	CONST robtarget p717:=[[0.0000,-127.8373,13.7328],[0.0000,-0.0467,0.9989,0.0000],[-1,0,-1,0],[9E+09,0.0000,-489.6442,9E+09,9E+09,9E+09]];
	CONST robtarget p718:=[[0.0000,-127.6671,13.7523],[0.0000,-0.0390,0.9992,0.0000],[-1,0,-1,0],[9E+09,0.0000,-490.5328,9E+09,9E+09,9E+09]];
	CONST robtarget p719:=[[0.0000,-127.5276,13.7719],[0.0000,-0.0312,0.9995,0.0000],[-1,0,-1,0],[9E+09,0.0000,-491.4237,9E+09,9E+09,9E+09]];
	CONST robtarget p720:=[[0.0000,-127.4190,13.7914],[0.0000,-0.0234,0.9997,0.0000],[-1,0,-1,0],[9E+09,0.0000,-492.3162,9E+09,9E+09,9E+09]];
	CONST robtarget p721:=[[0.0000,-127.3414,13.8109],[0.0000,-0.0156,0.9999,0.0000],[-1,0,-1,0],[9E+09,0.0000,-493.2101,9E+09,9E+09,9E+09]];
	CONST robtarget p722:=[[0.0000,-127.2948,13.8305],[0.0000,-0.0078,1.0000,0.0000],[-1,0,-1,0],[9E+09,0.0000,-494.1048,9E+09,9E+09,9E+09]];
	CONST robtarget p723:=[[0.0000,-127.2792,13.8500],[0.0000,-0.0000,-1.0000,0.0000],[-1,0,-1,0],[9E+09,0.0000,-495.0000,9E+09,9E+09,9E+09]];
	CONST robtarget p724:=[[0.0000,-127.2948,13.8695],[0.0000,-0.0078,-1.0000,0.0000],[-1,0,-1,0],[9E+09,0.0000,-495.8952,9E+09,9E+09,9E+09]];
	CONST robtarget p725:=[[0.0000,-127.3414,13.8891],[0.0000,-0.0156,-0.9999,0.0000],[-1,0,-1,0],[9E+09,0.0000,-496.7899,9E+09,9E+09,9E+09]];
	CONST robtarget p726:=[[0.0000,-127.4190,13.9086],[0.0000,-0.0234,-0.9997,0.0000],[-1,0,-1,0],[9E+09,0.0000,-497.6838,9E+09,9E+09,9E+09]];
	CONST robtarget p727:=[[0.0000,-127.5276,13.9281],[0.0000,-0.0312,-0.9995,0.0000],[-1,0,-1,0],[9E+09,0.0000,-498.5763,9E+09,9E+09,9E+09]];
	CONST robtarget p728:=[[0.0000,-127.6671,13.9477],[0.0000,-0.0390,-0.9992,0.0000],[-1,0,-1,0],[9E+09,0.0000,-499.4672,9E+09,9E+09,9E+09]];
	CONST robtarget p729:=[[0.0000,-127.8373,13.9672],[0.0000,-0.0467,-0.9989,0.0000],[-1,0,-1,0],[9E+09,0.0000,-500.3558,9E+09,9E+09,9E+09]];
	CONST robtarget p730:=[[0.0000,-128.0383,13.9867],[0.0000,-0.0544,-0.9985,0.0000],[-1,0,-1,0],[9E+09,0.0000,-501.2419,9E+09,9E+09,9E+09]];
	CONST robtarget p731:=[[0.0000,-128.2697,14.0062],[0.0000,-0.0621,-0.9981,0.0000],[-1,0,-1,0],[9E+09,0.0000,-502.1250,9E+09,9E+09,9E+09]];
	CONST robtarget p732:=[[0.0000,-128.5316,14.0258],[0.0000,-0.0698,-0.9976,0.0000],[-1,0,-1,0],[9E+09,0.0000,-503.0047,9E+09,9E+09,9E+09]];
	CONST robtarget p733:=[[0.0000,-128.8236,14.0453],[0.0000,-0.0774,-0.9970,0.0000],[-1,0,-1,0],[9E+09,0.0000,-503.8807,9E+09,9E+09,9E+09]];
	CONST robtarget p734:=[[0.0000,-129.1455,14.0648],[0.0000,-0.0850,-0.9964,0.0000],[-1,0,-1,0],[9E+09,0.0000,-504.7524,9E+09,9E+09,9E+09]];
	CONST robtarget p735:=[[0.0000,-129.4972,14.0844],[0.0000,-0.0925,-0.9957,0.0000],[-1,0,-1,0],[9E+09,0.0000,-505.6197,9E+09,9E+09,9E+09]];
	CONST robtarget p736:=[[0.0000,-129.8784,14.1039],[0.0000,-0.1000,-0.9950,0.0000],[-1,0,-1,0],[9E+09,0.0000,-506.4820,9E+09,9E+09,9E+09]];
	CONST robtarget p737:=[[0.0000,-130.2889,14.1234],[0.0000,-0.1075,-0.9942,0.0000],[-1,0,-1,0],[9E+09,0.0000,-507.3391,9E+09,9E+09,9E+09]];
	CONST robtarget p738:=[[0.0000,-130.7283,14.1430],[0.0000,-0.1149,-0.9934,0.0000],[-1,0,-1,0],[9E+09,0.0000,-508.1906,9E+09,9E+09,9E+09]];
	CONST robtarget p739:=[[0.0000,-131.1964,14.1625],[0.0000,-0.1222,-0.9925,0.0000],[-1,0,-1,0],[9E+09,0.0000,-509.0362,9E+09,9E+09,9E+09]];
	CONST robtarget p740:=[[0.0000,-131.6929,14.1820],[0.0000,-0.1295,-0.9916,0.0000],[-1,0,-1,0],[9E+09,0.0000,-509.8757,9E+09,9E+09,9E+09]];
	CONST robtarget p741:=[[0.0000,-132.2174,14.2016],[0.0000,-0.1367,-0.9906,0.0000],[-1,0,-1,0],[9E+09,0.0000,-510.7086,9E+09,9E+09,9E+09]];
	CONST robtarget p742:=[[0.0000,-132.7697,14.2211],[0.0000,-0.1438,-0.9896,0.0000],[-1,0,-1,0],[9E+09,0.0000,-511.5348,9E+09,9E+09,9E+09]];
	CONST robtarget p743:=[[0.0000,-133.3493,14.2406],[0.0000,-0.1509,-0.9886,0.0000],[-1,0,-1,0],[9E+09,0.0000,-512.3540,9E+09,9E+09,9E+09]];
	CONST robtarget p744:=[[0.0000,-133.9559,14.2602],[0.0000,-0.1579,-0.9875,0.0000],[-1,0,-1,0],[9E+09,0.0000,-513.1660,9E+09,9E+09,9E+09]];
	CONST robtarget p745:=[[0.0000,-134.5892,14.2797],[0.0000,-0.1648,-0.9863,0.0000],[-1,0,-1,0],[9E+09,0.0000,-513.9704,9E+09,9E+09,9E+09]];
	CONST robtarget p746:=[[0.0000,-135.2488,14.2992],[0.0000,-0.1716,-0.9852,0.0000],[-1,0,-1,0],[9E+09,0.0000,-514.7672,9E+09,9E+09,9E+09]];
	CONST robtarget p747:=[[0.0000,-135.9343,14.3187],[0.0000,-0.1784,-0.9840,0.0000],[-1,0,-1,0],[9E+09,0.0000,-515.5560,9E+09,9E+09,9E+09]];
	CONST robtarget p748:=[[0.0000,-136.6452,14.3383],[0.0000,-0.1851,-0.9827,0.0000],[-1,0,-1,0],[9E+09,0.0000,-516.3369,9E+09,9E+09,9E+09]];
	CONST robtarget p749:=[[0.0000,-137.3813,14.3578],[0.0000,-0.1917,-0.9814,0.0000],[-1,0,-1,0],[9E+09,0.0000,-517.1094,9E+09,9E+09,9E+09]];
	CONST robtarget p750:=[[0.0000,-138.1421,14.3773],[0.0000,-0.1983,-0.9801,0.0000],[-1,0,-1,0],[9E+09,0.0000,-517.8737,9E+09,9E+09,9E+09]];
	CONST robtarget p751:=[[0.0000,-138.9273,14.3969],[0.0000,-0.2047,-0.9788,0.0000],[-1,0,-1,0],[9E+09,0.0000,-518.6294,9E+09,9E+09,9E+09]];
	CONST robtarget p752:=[[0.0000,-139.7363,14.4164],[0.0000,-0.2111,-0.9775,0.0000],[-1,0,-1,0],[9E+09,0.0000,-519.3765,9E+09,9E+09,9E+09]];
	CONST robtarget p753:=[[0.0000,-140.5687,14.4359],[0.0000,-0.2174,-0.9761,0.0000],[-1,0,-1,0],[9E+09,0.0000,-520.1148,9E+09,9E+09,9E+09]];
	CONST robtarget p754:=[[0.0000,-141.4243,14.4555],[0.0000,-0.2236,-0.9747,0.0000],[-1,0,-1,0],[9E+09,0.0000,-520.8444,9E+09,9E+09,9E+09]];
	CONST robtarget p755:=[[0.0000,-142.3025,14.4750],[0.0000,-0.2298,-0.9732,0.0000],[-1,0,-1,0],[9E+09,0.0000,-521.5651,9E+09,9E+09,9E+09]];
	CONST robtarget p756:=[[0.0000,-143.2029,14.4945],[0.0000,-0.2358,-0.9718,0.0000],[-1,0,-1,0],[9E+09,0.0000,-522.2768,9E+09,9E+09,9E+09]];
	CONST robtarget p757:=[[0.0000,-144.1252,14.5141],[0.0000,-0.2417,-0.9703,0.0000],[-1,0,-1,0],[9E+09,0.0000,-522.9795,9E+09,9E+09,9E+09]];
	CONST robtarget p758:=[[0.0000,-145.0688,14.5336],[0.0000,-0.2476,-0.9689,0.0000],[-1,0,-1,0],[9E+09,0.0000,-523.6731,9E+09,9E+09,9E+09]];
	CONST robtarget p759:=[[0.0000,-146.0335,14.5531],[0.0000,-0.2534,-0.9674,0.0000],[-1,0,-1,0],[9E+09,0.0000,-524.3578,9E+09,9E+09,9E+09]];
	CONST robtarget p760:=[[0.0000,-147.0187,14.5727],[0.0000,-0.2591,-0.9659,0.0000],[-1,0,-1,0],[9E+09,0.0000,-525.0333,9E+09,9E+09,9E+09]];
	CONST robtarget p761:=[[0.0000,-148.0241,14.5922],[0.0000,-0.2647,-0.9643,0.0000],[-1,0,-1,0],[9E+09,0.0000,-525.6997,9E+09,9E+09,9E+09]];
	CONST robtarget p762:=[[0.0000,-149.0492,14.6117],[0.0000,-0.2702,-0.9628,0.0000],[-1,0,-1,0],[9E+09,0.0000,-526.3571,9E+09,9E+09,9E+09]];
	CONST robtarget p763:=[[0.0000,-150.0937,14.6312],[0.0000,-0.2757,-0.9612,0.0000],[-1,0,-1,0],[9E+09,0.0000,-527.0054,9E+09,9E+09,9E+09]];
	CONST robtarget p764:=[[0.0000,-151.1572,14.6508],[0.0000,-0.2810,-0.9597,0.0000],[-1,0,-1,0],[9E+09,0.0000,-527.6446,9E+09,9E+09,9E+09]];
	CONST robtarget p765:=[[0.0000,-152.2391,14.6703],[0.0000,-0.2863,-0.9581,0.0000],[-1,0,-1,0],[9E+09,0.0000,-528.2749,9E+09,9E+09,9E+09]];
	CONST robtarget p766:=[[0.0000,-153.3393,14.6898],[0.0000,-0.2915,-0.9566,0.0000],[-1,0,-1,0],[9E+09,0.0000,-528.8962,9E+09,9E+09,9E+09]];
	CONST robtarget p767:=[[0.0000,-154.4572,14.7094],[0.0000,-0.2966,-0.9550,0.0000],[-1,0,-1,0],[9E+09,0.0000,-529.5085,9E+09,9E+09,9E+09]];
	CONST robtarget p768:=[[0.0000,-155.5925,14.7289],[0.0000,-0.3016,-0.9534,0.0000],[-1,0,-1,0],[9E+09,0.0000,-530.1120,9E+09,9E+09,9E+09]];
	CONST robtarget p769:=[[0.0000,-156.7448,14.7484],[0.0000,-0.3066,-0.9518,0.0000],[-1,0,-1,0],[9E+09,0.0000,-530.7067,9E+09,9E+09,9E+09]];
	CONST robtarget p770:=[[0.0000,-157.9138,14.7680],[0.0000,-0.3114,-0.9503,0.0000],[-1,0,-1,0],[9E+09,0.0000,-531.2926,9E+09,9E+09,9E+09]];
	CONST robtarget p771:=[[0.0000,-159.0990,14.7875],[0.0000,-0.3162,-0.9487,0.0000],[-1,0,-1,0],[9E+09,0.0000,-531.8699,9E+09,9E+09,9E+09]];
	CONST robtarget p772:=[[0.0000,-160.3002,14.8070],[0.0000,-0.3209,-0.9471,0.0000],[-1,0,-1,0],[9E+09,0.0000,-532.4386,9E+09,9E+09,9E+09]];
	CONST robtarget p773:=[[0.0000,-161.5169,14.8266],[0.0000,-0.3256,-0.9455,0.0000],[-1,0,-1,0],[9E+09,0.0000,-532.9987,9E+09,9E+09,9E+09]];
	CONST robtarget p774:=[[0.0000,-162.7488,14.8461],[0.0000,-0.3301,-0.9439,0.0000],[-1,0,-1,0],[9E+09,0.0000,-533.5505,9E+09,9E+09,9E+09]];
	CONST robtarget p775:=[[0.0000,-163.9955,14.8656],[0.0000,-0.3346,-0.9424,0.0000],[-1,0,-1,0],[9E+09,0.0000,-534.0939,9E+09,9E+09,9E+09]];
	CONST robtarget p776:=[[0.0000,-165.2568,14.8852],[0.0000,-0.3390,-0.9408,0.0000],[-1,0,-1,0],[9E+09,0.0000,-534.6290,9E+09,9E+09,9E+09]];
	CONST robtarget p777:=[[0.0000,-166.5323,14.9047],[0.0000,-0.3433,-0.9392,0.0000],[-1,0,-1,0],[9E+09,0.0000,-535.1560,9E+09,9E+09,9E+09]];
	CONST robtarget p778:=[[0.0000,-167.8217,14.9242],[0.0000,-0.3475,-0.9377,0.0000],[-1,0,-1,0],[9E+09,0.0000,-535.6749,9E+09,9E+09,9E+09]];
	CONST robtarget p779:=[[0.0000,-169.1246,14.9437],[0.0000,-0.3517,-0.9361,0.0000],[-1,0,-1,0],[9E+09,0.0000,-536.1859,9E+09,9E+09,9E+09]];
	CONST robtarget p780:=[[0.0000,-170.4407,14.9633],[0.0000,-0.3558,-0.9345,0.0000],[-1,0,-1,0],[9E+09,0.0000,-536.6891,9E+09,9E+09,9E+09]];
	CONST robtarget p781:=[[0.0000,-171.7699,14.9828],[0.0000,-0.3599,-0.9330,0.0000],[-1,0,-1,0],[9E+09,0.0000,-537.1844,9E+09,9E+09,9E+09]];
	CONST robtarget p782:=[[0.0000,-173.1116,15.0023],[0.0000,-0.3638,-0.9315,0.0000],[-1,0,-1,0],[9E+09,0.0000,-537.6722,9E+09,9E+09,9E+09]];
	CONST robtarget p783:=[[0.0000,-174.4657,15.0219],[0.0000,-0.3677,-0.9299,0.0000],[-1,0,-1,0],[9E+09,0.0000,-538.1524,9E+09,9E+09,9E+09]];
	CONST robtarget p784:=[[0.0000,-175.8319,15.0414],[0.0000,-0.3716,-0.9284,0.0000],[-1,0,-1,0],[9E+09,0.0000,-538.6252,9E+09,9E+09,9E+09]];
	CONST robtarget p785:=[[0.0000,-177.2098,15.0609],[0.0000,-0.3753,-0.9269,0.0000],[-1,0,-1,0],[9E+09,0.0000,-539.0906,9E+09,9E+09,9E+09]];
	CONST robtarget p786:=[[0.0000,-178.5993,15.0805],[0.0000,-0.3790,-0.9254,0.0000],[-1,0,-1,0],[9E+09,0.0000,-539.5489,9E+09,9E+09,9E+09]];
	CONST robtarget p787:=[[0.0000,-180.0000,15.1000],[0.0000,-0.3827,0.9239,0.0000],[-1,0,-1,0],[9E+09,0.0000,-540.0000,9E+09,9E+09,9E+09]];
	CONST robtarget p788:=[[0.0000,-178.5993,15.1195],[0.0000,-0.3790,0.9254,0.0000],[-1,0,-1,0],[9E+09,0.0000,-540.4511,9E+09,9E+09,9E+09]];
	CONST robtarget p789:=[[0.0000,-177.2098,15.1391],[0.0000,-0.3753,0.9269,0.0000],[-1,0,-1,0],[9E+09,0.0000,-540.9094,9E+09,9E+09,9E+09]];
	CONST robtarget p790:=[[0.0000,-175.8319,15.1586],[0.0000,-0.3716,0.9284,0.0000],[-1,0,-1,0],[9E+09,0.0000,-541.3748,9E+09,9E+09,9E+09]];
	CONST robtarget p791:=[[0.0000,-174.4657,15.1781],[0.0000,-0.3677,0.9299,0.0000],[-1,0,-1,0],[9E+09,0.0000,-541.8476,9E+09,9E+09,9E+09]];
	CONST robtarget p792:=[[0.0000,-173.1116,15.1977],[0.0000,-0.3638,0.9315,0.0000],[-1,0,-1,0],[9E+09,0.0000,-542.3278,9E+09,9E+09,9E+09]];
	CONST robtarget p793:=[[0.0000,-171.7699,15.2172],[0.0000,-0.3599,0.9330,0.0000],[-1,0,-1,0],[9E+09,0.0000,-542.8156,9E+09,9E+09,9E+09]];
	CONST robtarget p794:=[[0.0000,-170.4407,15.2367],[0.0000,-0.3558,0.9345,0.0000],[-1,0,-1,0],[9E+09,0.0000,-543.3109,9E+09,9E+09,9E+09]];
	CONST robtarget p795:=[[0.0000,-169.1246,15.2562],[0.0000,-0.3517,0.9361,0.0000],[-1,0,-1,0],[9E+09,0.0000,-543.8141,9E+09,9E+09,9E+09]];
	CONST robtarget p796:=[[0.0000,-167.8217,15.2758],[0.0000,-0.3475,0.9377,0.0000],[-1,0,-1,0],[9E+09,0.0000,-544.3251,9E+09,9E+09,9E+09]];
	CONST robtarget p797:=[[0.0000,-166.5323,15.2953],[0.0000,-0.3433,0.9392,0.0000],[-1,0,-1,0],[9E+09,0.0000,-544.8440,9E+09,9E+09,9E+09]];
	CONST robtarget p798:=[[0.0000,-165.2568,15.3148],[0.0000,-0.3390,0.9408,0.0000],[-1,0,-1,0],[9E+09,0.0000,-545.3710,9E+09,9E+09,9E+09]];
	CONST robtarget p799:=[[0.0000,-163.9955,15.3344],[0.0000,-0.3346,0.9424,0.0000],[-1,0,-1,0],[9E+09,0.0000,-545.9061,9E+09,9E+09,9E+09]];
	CONST robtarget p800:=[[0.0000,-162.7488,15.3539],[0.0000,-0.3301,0.9439,0.0000],[-1,0,-1,0],[9E+09,0.0000,-546.4495,9E+09,9E+09,9E+09]];
	CONST robtarget p801:=[[0.0000,-161.5169,15.3734],[0.0000,-0.3256,0.9455,0.0000],[-1,0,-1,0],[9E+09,0.0000,-547.0013,9E+09,9E+09,9E+09]];
	CONST robtarget p802:=[[0.0000,-160.3002,15.3930],[0.0000,-0.3209,0.9471,0.0000],[-1,0,-1,0],[9E+09,0.0000,-547.5614,9E+09,9E+09,9E+09]];
	CONST robtarget p803:=[[0.0000,-159.0990,15.4125],[0.0000,-0.3162,0.9487,0.0000],[-1,0,-1,0],[9E+09,0.0000,-548.1301,9E+09,9E+09,9E+09]];
	CONST robtarget p804:=[[0.0000,-157.9138,15.4320],[0.0000,-0.3114,0.9503,0.0000],[-1,0,-1,0],[9E+09,0.0000,-548.7074,9E+09,9E+09,9E+09]];
	CONST robtarget p805:=[[0.0000,-156.7448,15.4516],[0.0000,-0.3066,0.9518,0.0000],[-1,0,-1,0],[9E+09,0.0000,-549.2933,9E+09,9E+09,9E+09]];
	CONST robtarget p806:=[[0.0000,-155.5925,15.4711],[0.0000,-0.3016,0.9534,0.0000],[-1,0,-1,0],[9E+09,0.0000,-549.8880,9E+09,9E+09,9E+09]];
	CONST robtarget p807:=[[0.0000,-154.4572,15.4906],[0.0000,-0.2966,0.9550,0.0000],[-1,0,-1,0],[9E+09,0.0000,-550.4915,9E+09,9E+09,9E+09]];
	CONST robtarget p808:=[[0.0000,-153.3393,15.5102],[0.0000,-0.2915,0.9566,0.0000],[-1,0,-1,0],[9E+09,0.0000,-551.1038,9E+09,9E+09,9E+09]];
	CONST robtarget p809:=[[0.0000,-152.2391,15.5297],[0.0000,-0.2863,0.9581,0.0000],[-1,0,-1,0],[9E+09,0.0000,-551.7251,9E+09,9E+09,9E+09]];
	CONST robtarget p810:=[[0.0000,-151.1572,15.5492],[0.0000,-0.2810,0.9597,0.0000],[-1,0,-1,0],[9E+09,0.0000,-552.3554,9E+09,9E+09,9E+09]];
	CONST robtarget p811:=[[0.0000,-150.0937,15.5687],[0.0000,-0.2757,0.9612,0.0000],[-1,0,-1,0],[9E+09,0.0000,-552.9946,9E+09,9E+09,9E+09]];
	CONST robtarget p812:=[[0.0000,-149.0492,15.5883],[0.0000,-0.2702,0.9628,0.0000],[-1,0,-1,0],[9E+09,0.0000,-553.6429,9E+09,9E+09,9E+09]];
	CONST robtarget p813:=[[0.0000,-148.0241,15.6078],[0.0000,-0.2647,0.9643,0.0000],[-1,0,-1,0],[9E+09,0.0000,-554.3003,9E+09,9E+09,9E+09]];
	CONST robtarget p814:=[[0.0000,-147.0187,15.6273],[0.0000,-0.2591,0.9659,0.0000],[-1,0,-1,0],[9E+09,0.0000,-554.9667,9E+09,9E+09,9E+09]];
	CONST robtarget p815:=[[0.0000,-146.0335,15.6469],[0.0000,-0.2534,0.9674,0.0000],[-1,0,-1,0],[9E+09,0.0000,-555.6422,9E+09,9E+09,9E+09]];
	CONST robtarget p816:=[[0.0000,-145.0688,15.6664],[0.0000,-0.2476,0.9689,0.0000],[-1,0,-1,0],[9E+09,0.0000,-556.3269,9E+09,9E+09,9E+09]];
	CONST robtarget p817:=[[0.0000,-144.1252,15.6859],[0.0000,-0.2417,0.9703,0.0000],[-1,0,-1,0],[9E+09,0.0000,-557.0205,9E+09,9E+09,9E+09]];
	CONST robtarget p818:=[[0.0000,-143.2029,15.7055],[0.0000,-0.2358,0.9718,0.0000],[-1,0,-1,0],[9E+09,0.0000,-557.7232,9E+09,9E+09,9E+09]];
	CONST robtarget p819:=[[0.0000,-142.3025,15.7250],[0.0000,-0.2298,0.9732,0.0000],[-1,0,-1,0],[9E+09,0.0000,-558.4349,9E+09,9E+09,9E+09]];
	CONST robtarget p820:=[[0.0000,-141.4243,15.7445],[0.0000,-0.2236,0.9747,0.0000],[-1,0,-1,0],[9E+09,0.0000,-559.1556,9E+09,9E+09,9E+09]];
	CONST robtarget p821:=[[0.0000,-140.5687,15.7641],[0.0000,-0.2174,0.9761,0.0000],[-1,0,-1,0],[9E+09,0.0000,-559.8852,9E+09,9E+09,9E+09]];
	CONST robtarget p822:=[[0.0000,-139.7363,15.7836],[0.0000,-0.2111,0.9775,0.0000],[-1,0,-1,0],[9E+09,0.0000,-560.6235,9E+09,9E+09,9E+09]];
	CONST robtarget p823:=[[0.0000,-138.9273,15.8031],[0.0000,-0.2047,0.9788,0.0000],[-1,0,-1,0],[9E+09,0.0000,-561.3706,9E+09,9E+09,9E+09]];
	CONST robtarget p824:=[[0.0000,-138.1421,15.8227],[0.0000,-0.1983,0.9801,0.0000],[-1,0,-1,0],[9E+09,0.0000,-562.1263,9E+09,9E+09,9E+09]];
	CONST robtarget p825:=[[0.0000,-137.3813,15.8422],[0.0000,-0.1917,0.9814,0.0000],[-1,0,-1,0],[9E+09,0.0000,-562.8906,9E+09,9E+09,9E+09]];
	CONST robtarget p826:=[[0.0000,-136.6452,15.8617],[0.0000,-0.1851,0.9827,0.0000],[-1,0,-1,0],[9E+09,0.0000,-563.6631,9E+09,9E+09,9E+09]];
	CONST robtarget p827:=[[0.0000,-135.9343,15.8812],[0.0000,-0.1784,0.9840,0.0000],[-1,0,-1,0],[9E+09,0.0000,-564.4440,9E+09,9E+09,9E+09]];
	CONST robtarget p828:=[[0.0000,-135.2488,15.9008],[0.0000,-0.1716,0.9852,0.0000],[-1,0,-1,0],[9E+09,0.0000,-565.2328,9E+09,9E+09,9E+09]];
	CONST robtarget p829:=[[0.0000,-134.5892,15.9203],[0.0000,-0.1648,0.9863,0.0000],[-1,0,-1,0],[9E+09,0.0000,-566.0296,9E+09,9E+09,9E+09]];
	CONST robtarget p830:=[[0.0000,-133.9559,15.9398],[0.0000,-0.1579,0.9875,0.0000],[-1,0,-1,0],[9E+09,0.0000,-566.8340,9E+09,9E+09,9E+09]];
	CONST robtarget p831:=[[0.0000,-133.3493,15.9594],[0.0000,-0.1509,0.9886,0.0000],[-1,0,-1,0],[9E+09,0.0000,-567.6460,9E+09,9E+09,9E+09]];
	CONST robtarget p832:=[[0.0000,-132.7697,15.9789],[0.0000,-0.1438,0.9896,0.0000],[-1,0,-1,0],[9E+09,0.0000,-568.4652,9E+09,9E+09,9E+09]];
	CONST robtarget p833:=[[0.0000,-132.2174,15.9984],[0.0000,-0.1367,0.9906,0.0000],[-1,0,-1,0],[9E+09,0.0000,-569.2914,9E+09,9E+09,9E+09]];
	CONST robtarget p834:=[[0.0000,-131.6929,16.0180],[0.0000,-0.1295,0.9916,0.0000],[-1,0,-1,0],[9E+09,0.0000,-570.1243,9E+09,9E+09,9E+09]];
	CONST robtarget p835:=[[0.0000,-131.1964,16.0375],[0.0000,-0.1222,0.9925,0.0000],[-1,0,-1,0],[9E+09,0.0000,-570.9638,9E+09,9E+09,9E+09]];
	CONST robtarget p836:=[[0.0000,-130.7283,16.0570],[0.0000,-0.1149,0.9934,0.0000],[-1,0,-1,0],[9E+09,0.0000,-571.8094,9E+09,9E+09,9E+09]];
	CONST robtarget p837:=[[0.0000,-130.2889,16.0766],[0.0000,-0.1075,0.9942,0.0000],[-1,0,-1,0],[9E+09,0.0000,-572.6609,9E+09,9E+09,9E+09]];
	CONST robtarget p838:=[[0.0000,-129.8784,16.0961],[0.0000,-0.1000,0.9950,0.0000],[-1,0,-1,0],[9E+09,0.0000,-573.5180,9E+09,9E+09,9E+09]];
	CONST robtarget p839:=[[0.0000,-129.4972,16.1156],[0.0000,-0.0925,0.9957,0.0000],[-1,0,-1,0],[9E+09,0.0000,-574.3803,9E+09,9E+09,9E+09]];
	CONST robtarget p840:=[[0.0000,-129.1455,16.1352],[0.0000,-0.0850,0.9964,0.0000],[-1,0,-1,0],[9E+09,0.0000,-575.2476,9E+09,9E+09,9E+09]];
	CONST robtarget p841:=[[0.0000,-128.8236,16.1547],[0.0000,-0.0774,0.9970,0.0000],[-1,0,-1,0],[9E+09,0.0000,-576.1193,9E+09,9E+09,9E+09]];
	CONST robtarget p842:=[[0.0000,-128.5316,16.1742],[0.0000,-0.0698,0.9976,0.0000],[-1,0,-1,0],[9E+09,0.0000,-576.9953,9E+09,9E+09,9E+09]];
	CONST robtarget p843:=[[0.0000,-128.2697,16.1938],[0.0000,-0.0621,0.9981,0.0000],[-1,0,-1,0],[9E+09,0.0000,-577.8750,9E+09,9E+09,9E+09]];
	CONST robtarget p844:=[[0.0000,-128.0383,16.2133],[0.0000,-0.0544,0.9985,0.0000],[-1,0,-1,0],[9E+09,0.0000,-578.7581,9E+09,9E+09,9E+09]];
	CONST robtarget p845:=[[0.0000,-127.8373,16.2328],[0.0000,-0.0467,0.9989,0.0000],[-1,0,-1,0],[9E+09,0.0000,-579.6442,9E+09,9E+09,9E+09]];
	CONST robtarget p846:=[[0.0000,-127.6671,16.2523],[0.0000,-0.0390,0.9992,0.0000],[-1,0,-1,0],[9E+09,0.0000,-580.5328,9E+09,9E+09,9E+09]];
	CONST robtarget p847:=[[0.0000,-127.5276,16.2719],[0.0000,-0.0312,0.9995,0.0000],[-1,0,-1,0],[9E+09,0.0000,-581.4237,9E+09,9E+09,9E+09]];
	CONST robtarget p848:=[[0.0000,-127.4190,16.2914],[0.0000,-0.0234,0.9997,0.0000],[-1,0,-1,0],[9E+09,0.0000,-582.3162,9E+09,9E+09,9E+09]];
	CONST robtarget p849:=[[0.0000,-127.3414,16.3109],[0.0000,-0.0156,0.9999,0.0000],[-1,0,-1,0],[9E+09,0.0000,-583.2101,9E+09,9E+09,9E+09]];
	CONST robtarget p850:=[[0.0000,-127.2948,16.3305],[0.0000,-0.0078,1.0000,0.0000],[-1,0,-1,0],[9E+09,0.0000,-584.1048,9E+09,9E+09,9E+09]];
	CONST robtarget p851:=[[0.0000,-127.2792,16.3500],[0.0000,0.0000,1.0000,0.0000],[-1,0,-1,0],[9E+09,0.0000,-585.0000,9E+09,9E+09,9E+09]];
	CONST robtarget p852:=[[0.0000,-127.2948,16.3695],[0.0000,-0.0078,-1.0000,0.0000],[-1,0,-1,0],[9E+09,0.0000,-585.8952,9E+09,9E+09,9E+09]];
	CONST robtarget p853:=[[0.0000,-127.3414,16.3891],[0.0000,-0.0156,-0.9999,0.0000],[-1,0,-1,0],[9E+09,0.0000,-586.7899,9E+09,9E+09,9E+09]];
	CONST robtarget p854:=[[0.0000,-127.4190,16.4086],[0.0000,-0.0234,-0.9997,0.0000],[-1,0,-1,0],[9E+09,0.0000,-587.6838,9E+09,9E+09,9E+09]];
	CONST robtarget p855:=[[0.0000,-127.5276,16.4281],[0.0000,-0.0312,-0.9995,0.0000],[-1,0,-1,0],[9E+09,0.0000,-588.5763,9E+09,9E+09,9E+09]];
	CONST robtarget p856:=[[0.0000,-127.6671,16.4477],[0.0000,-0.0390,-0.9992,0.0000],[-1,0,-1,0],[9E+09,0.0000,-589.4672,9E+09,9E+09,9E+09]];
	CONST robtarget p857:=[[0.0000,-127.8373,16.4672],[0.0000,-0.0467,-0.9989,0.0000],[-1,0,-1,0],[9E+09,0.0000,-590.3558,9E+09,9E+09,9E+09]];
	CONST robtarget p858:=[[0.0000,-128.0383,16.4867],[0.0000,-0.0544,-0.9985,0.0000],[-1,0,-1,0],[9E+09,0.0000,-591.2419,9E+09,9E+09,9E+09]];
	CONST robtarget p859:=[[0.0000,-128.2697,16.5063],[0.0000,-0.0621,-0.9981,0.0000],[-1,0,-1,0],[9E+09,0.0000,-592.1250,9E+09,9E+09,9E+09]];
	CONST robtarget p860:=[[0.0000,-128.5316,16.5258],[0.0000,-0.0698,-0.9976,0.0000],[-1,0,-1,0],[9E+09,0.0000,-593.0047,9E+09,9E+09,9E+09]];
	CONST robtarget p861:=[[0.0000,-128.8236,16.5453],[0.0000,-0.0774,-0.9970,0.0000],[-1,0,-1,0],[9E+09,0.0000,-593.8807,9E+09,9E+09,9E+09]];
	CONST robtarget p862:=[[0.0000,-129.1455,16.5648],[0.0000,-0.0850,-0.9964,0.0000],[-1,0,-1,0],[9E+09,0.0000,-594.7524,9E+09,9E+09,9E+09]];
	CONST robtarget p863:=[[0.0000,-129.4972,16.5844],[0.0000,-0.0925,-0.9957,0.0000],[-1,0,-1,0],[9E+09,0.0000,-595.6197,9E+09,9E+09,9E+09]];
	CONST robtarget p864:=[[0.0000,-129.8784,16.6039],[0.0000,-0.1000,-0.9950,0.0000],[-1,0,-1,0],[9E+09,0.0000,-596.4820,9E+09,9E+09,9E+09]];
	CONST robtarget p865:=[[0.0000,-130.2889,16.6234],[0.0000,-0.1075,-0.9942,0.0000],[-1,0,-1,0],[9E+09,0.0000,-597.3391,9E+09,9E+09,9E+09]];
	CONST robtarget p866:=[[0.0000,-130.7283,16.6430],[0.0000,-0.1149,-0.9934,0.0000],[-1,0,-1,0],[9E+09,0.0000,-598.1906,9E+09,9E+09,9E+09]];
	CONST robtarget p867:=[[0.0000,-131.1964,16.6625],[0.0000,-0.1222,-0.9925,0.0000],[-1,0,-1,0],[9E+09,0.0000,-599.0362,9E+09,9E+09,9E+09]];
	CONST robtarget p868:=[[0.0000,-131.6929,16.6820],[0.0000,-0.1295,-0.9916,0.0000],[-1,0,-1,0],[9E+09,0.0000,-599.8757,9E+09,9E+09,9E+09]];
	CONST robtarget p869:=[[0.0000,-132.2174,16.7016],[0.0000,-0.1367,-0.9906,0.0000],[-1,0,-1,0],[9E+09,0.0000,-600.7086,9E+09,9E+09,9E+09]];
	CONST robtarget p870:=[[0.0000,-132.7697,16.7211],[0.0000,-0.1438,-0.9896,0.0000],[-1,0,-1,0],[9E+09,0.0000,-601.5348,9E+09,9E+09,9E+09]];
	CONST robtarget p871:=[[0.0000,-133.3493,16.7406],[0.0000,-0.1509,-0.9886,0.0000],[-1,0,-1,0],[9E+09,0.0000,-602.3540,9E+09,9E+09,9E+09]];
	CONST robtarget p872:=[[0.0000,-133.9559,16.7602],[0.0000,-0.1579,-0.9875,0.0000],[-1,0,-1,0],[9E+09,0.0000,-603.1660,9E+09,9E+09,9E+09]];
	CONST robtarget p873:=[[0.0000,-134.5892,16.7797],[0.0000,-0.1648,-0.9863,0.0000],[-1,0,-1,0],[9E+09,0.0000,-603.9704,9E+09,9E+09,9E+09]];
	CONST robtarget p874:=[[0.0000,-135.2488,16.7992],[0.0000,-0.1716,-0.9852,0.0000],[-1,0,-1,0],[9E+09,0.0000,-604.7672,9E+09,9E+09,9E+09]];
	CONST robtarget p875:=[[0.0000,-135.9343,16.8188],[0.0000,-0.1784,-0.9840,0.0000],[-1,0,-1,0],[9E+09,0.0000,-605.5560,9E+09,9E+09,9E+09]];
	CONST robtarget p876:=[[0.0000,-136.6452,16.8383],[0.0000,-0.1851,-0.9827,0.0000],[-1,0,-1,0],[9E+09,0.0000,-606.3369,9E+09,9E+09,9E+09]];
	CONST robtarget p877:=[[0.0000,-137.3813,16.8578],[0.0000,-0.1917,-0.9814,0.0000],[-1,0,-1,0],[9E+09,0.0000,-607.1094,9E+09,9E+09,9E+09]];
	CONST robtarget p878:=[[0.0000,-138.1421,16.8773],[0.0000,-0.1983,-0.9801,0.0000],[-1,0,-1,0],[9E+09,0.0000,-607.8737,9E+09,9E+09,9E+09]];
	CONST robtarget p879:=[[0.0000,-138.9273,16.8969],[0.0000,-0.2047,-0.9788,0.0000],[-1,0,-1,0],[9E+09,0.0000,-608.6294,9E+09,9E+09,9E+09]];
	CONST robtarget p880:=[[0.0000,-139.7363,16.9164],[0.0000,-0.2111,-0.9775,0.0000],[-1,0,-1,0],[9E+09,0.0000,-609.3765,9E+09,9E+09,9E+09]];
	CONST robtarget p881:=[[0.0000,-140.5687,16.9359],[0.0000,-0.2174,-0.9761,0.0000],[-1,0,-1,0],[9E+09,0.0000,-610.1148,9E+09,9E+09,9E+09]];
	CONST robtarget p882:=[[0.0000,-141.4243,16.9555],[0.0000,-0.2236,-0.9747,0.0000],[-1,0,-1,0],[9E+09,0.0000,-610.8444,9E+09,9E+09,9E+09]];
	CONST robtarget p883:=[[0.0000,-142.3025,16.9750],[0.0000,-0.2298,-0.9732,0.0000],[-1,0,-1,0],[9E+09,0.0000,-611.5651,9E+09,9E+09,9E+09]];
	CONST robtarget p884:=[[0.0000,-143.2029,16.9945],[0.0000,-0.2358,-0.9718,0.0000],[-1,0,-1,0],[9E+09,0.0000,-612.2768,9E+09,9E+09,9E+09]];
	CONST robtarget p885:=[[0.0000,-144.1252,17.0141],[0.0000,-0.2417,-0.9703,0.0000],[-1,0,-1,0],[9E+09,0.0000,-612.9795,9E+09,9E+09,9E+09]];
	CONST robtarget p886:=[[0.0000,-145.0688,17.0336],[0.0000,-0.2476,-0.9689,0.0000],[-1,0,-1,0],[9E+09,0.0000,-613.6731,9E+09,9E+09,9E+09]];
	CONST robtarget p887:=[[0.0000,-146.0335,17.0531],[0.0000,-0.2534,-0.9674,0.0000],[-1,0,-1,0],[9E+09,0.0000,-614.3578,9E+09,9E+09,9E+09]];
	CONST robtarget p888:=[[0.0000,-147.0187,17.0727],[0.0000,-0.2591,-0.9659,0.0000],[-1,0,-1,0],[9E+09,0.0000,-615.0333,9E+09,9E+09,9E+09]];
	CONST robtarget p889:=[[0.0000,-148.0241,17.0922],[0.0000,-0.2647,-0.9643,0.0000],[-1,0,-1,0],[9E+09,0.0000,-615.6997,9E+09,9E+09,9E+09]];
	CONST robtarget p890:=[[0.0000,-149.0492,17.1117],[0.0000,-0.2702,-0.9628,0.0000],[-1,0,-1,0],[9E+09,0.0000,-616.3571,9E+09,9E+09,9E+09]];
	CONST robtarget p891:=[[0.0000,-150.0937,17.1313],[0.0000,-0.2757,-0.9612,0.0000],[-1,0,-1,0],[9E+09,0.0000,-617.0054,9E+09,9E+09,9E+09]];
	CONST robtarget p892:=[[0.0000,-151.1572,17.1508],[0.0000,-0.2810,-0.9597,0.0000],[-1,0,-1,0],[9E+09,0.0000,-617.6446,9E+09,9E+09,9E+09]];
	CONST robtarget p893:=[[0.0000,-152.2391,17.1703],[0.0000,-0.2863,-0.9581,0.0000],[-1,0,-1,0],[9E+09,0.0000,-618.2749,9E+09,9E+09,9E+09]];
	CONST robtarget p894:=[[0.0000,-153.3393,17.1898],[0.0000,-0.2915,-0.9566,0.0000],[-1,0,-1,0],[9E+09,0.0000,-618.8962,9E+09,9E+09,9E+09]];
	CONST robtarget p895:=[[0.0000,-154.4572,17.2094],[0.0000,-0.2966,-0.9550,0.0000],[-1,0,-1,0],[9E+09,0.0000,-619.5085,9E+09,9E+09,9E+09]];
	CONST robtarget p896:=[[0.0000,-155.5925,17.2289],[0.0000,-0.3016,-0.9534,0.0000],[-1,0,-1,0],[9E+09,0.0000,-620.1120,9E+09,9E+09,9E+09]];
	CONST robtarget p897:=[[0.0000,-156.7448,17.2484],[0.0000,-0.3066,-0.9518,0.0000],[-1,0,-1,0],[9E+09,0.0000,-620.7067,9E+09,9E+09,9E+09]];
	CONST robtarget p898:=[[0.0000,-157.9138,17.2680],[0.0000,-0.3114,-0.9503,0.0000],[-1,0,-1,0],[9E+09,0.0000,-621.2926,9E+09,9E+09,9E+09]];
	CONST robtarget p899:=[[0.0000,-159.0990,17.2875],[0.0000,-0.3162,-0.9487,0.0000],[-1,0,-1,0],[9E+09,0.0000,-621.8699,9E+09,9E+09,9E+09]];
	CONST robtarget p900:=[[0.0000,-160.3002,17.3070],[0.0000,-0.3209,-0.9471,0.0000],[-1,0,-1,0],[9E+09,0.0000,-622.4386,9E+09,9E+09,9E+09]];
	CONST robtarget p901:=[[0.0000,-161.5169,17.3266],[0.0000,-0.3256,-0.9455,0.0000],[-1,0,-1,0],[9E+09,0.0000,-622.9987,9E+09,9E+09,9E+09]];
	CONST robtarget p902:=[[0.0000,-162.7488,17.3461],[0.0000,-0.3301,-0.9439,0.0000],[-1,0,-1,0],[9E+09,0.0000,-623.5505,9E+09,9E+09,9E+09]];
	CONST robtarget p903:=[[0.0000,-163.9955,17.3656],[0.0000,-0.3346,-0.9424,0.0000],[-1,0,-1,0],[9E+09,0.0000,-624.0939,9E+09,9E+09,9E+09]];
	CONST robtarget p904:=[[0.0000,-165.2568,17.3852],[0.0000,-0.3390,-0.9408,0.0000],[-1,0,-1,0],[9E+09,0.0000,-624.6290,9E+09,9E+09,9E+09]];
	CONST robtarget p905:=[[0.0000,-166.5323,17.4047],[0.0000,-0.3433,-0.9392,0.0000],[-1,0,-1,0],[9E+09,0.0000,-625.1560,9E+09,9E+09,9E+09]];
	CONST robtarget p906:=[[0.0000,-167.8217,17.4242],[0.0000,-0.3475,-0.9377,0.0000],[-1,0,-1,0],[9E+09,0.0000,-625.6749,9E+09,9E+09,9E+09]];
	CONST robtarget p907:=[[0.0000,-169.1246,17.4438],[0.0000,-0.3517,-0.9361,0.0000],[-1,0,-1,0],[9E+09,0.0000,-626.1859,9E+09,9E+09,9E+09]];
	CONST robtarget p908:=[[0.0000,-170.4407,17.4633],[0.0000,-0.3558,-0.9345,0.0000],[-1,0,-1,0],[9E+09,0.0000,-626.6891,9E+09,9E+09,9E+09]];
	CONST robtarget p909:=[[0.0000,-171.7699,17.4828],[0.0000,-0.3599,-0.9330,0.0000],[-1,0,-1,0],[9E+09,0.0000,-627.1844,9E+09,9E+09,9E+09]];
	CONST robtarget p910:=[[0.0000,-173.1116,17.5023],[0.0000,-0.3638,-0.9315,0.0000],[-1,0,-1,0],[9E+09,0.0000,-627.6722,9E+09,9E+09,9E+09]];
	CONST robtarget p911:=[[0.0000,-174.4657,17.5219],[0.0000,-0.3677,-0.9299,0.0000],[-1,0,-1,0],[9E+09,0.0000,-628.1524,9E+09,9E+09,9E+09]];
	CONST robtarget p912:=[[0.0000,-175.8319,17.5414],[0.0000,-0.3716,-0.9284,0.0000],[-1,0,-1,0],[9E+09,0.0000,-628.6252,9E+09,9E+09,9E+09]];
	CONST robtarget p913:=[[0.0000,-177.2098,17.5609],[0.0000,-0.3753,-0.9269,0.0000],[-1,0,-1,0],[9E+09,0.0000,-629.0906,9E+09,9E+09,9E+09]];
	CONST robtarget p914:=[[0.0000,-178.5993,17.5805],[0.0000,-0.3790,-0.9254,0.0000],[-1,0,-1,0],[9E+09,0.0000,-629.5489,9E+09,9E+09,9E+09]];
	CONST robtarget p915:=[[0.0000,-180.0000,17.6000],[0.0000,-0.3827,0.9239,0.0000],[-1,0,-1,0],[9E+09,0.0000,-630.0000,9E+09,9E+09,9E+09]];
	CONST robtarget p916:=[[0.0000,-178.5993,17.6195],[0.0000,-0.3790,0.9254,0.0000],[-1,0,-1,0],[9E+09,0.0000,-630.4511,9E+09,9E+09,9E+09]];
	CONST robtarget p917:=[[0.0000,-177.2098,17.6391],[0.0000,-0.3753,0.9269,0.0000],[-1,0,-1,0],[9E+09,0.0000,-630.9094,9E+09,9E+09,9E+09]];
	CONST robtarget p918:=[[0.0000,-175.8319,17.6586],[0.0000,-0.3716,0.9284,0.0000],[-1,0,-1,0],[9E+09,0.0000,-631.3748,9E+09,9E+09,9E+09]];
	CONST robtarget p919:=[[0.0000,-174.4657,17.6781],[0.0000,-0.3677,0.9299,0.0000],[-1,0,-1,0],[9E+09,0.0000,-631.8476,9E+09,9E+09,9E+09]];
	CONST robtarget p920:=[[0.0000,-173.1116,17.6977],[0.0000,-0.3638,0.9315,0.0000],[-1,0,-1,0],[9E+09,0.0000,-632.3278,9E+09,9E+09,9E+09]];
	CONST robtarget p921:=[[0.0000,-171.7699,17.7172],[0.0000,-0.3599,0.9330,0.0000],[-1,0,-1,0],[9E+09,0.0000,-632.8156,9E+09,9E+09,9E+09]];
	CONST robtarget p922:=[[0.0000,-170.4407,17.7367],[0.0000,-0.3558,0.9345,0.0000],[-1,0,-1,0],[9E+09,0.0000,-633.3109,9E+09,9E+09,9E+09]];
	CONST robtarget p923:=[[0.0000,-169.1246,17.7563],[0.0000,-0.3517,0.9361,0.0000],[-1,0,-1,0],[9E+09,0.0000,-633.8141,9E+09,9E+09,9E+09]];
	CONST robtarget p924:=[[0.0000,-167.8217,17.7758],[0.0000,-0.3475,0.9377,0.0000],[-1,0,-1,0],[9E+09,0.0000,-634.3251,9E+09,9E+09,9E+09]];
	CONST robtarget p925:=[[0.0000,-166.5323,17.7953],[0.0000,-0.3433,0.9392,0.0000],[-1,0,-1,0],[9E+09,0.0000,-634.8440,9E+09,9E+09,9E+09]];
	CONST robtarget p926:=[[0.0000,-165.2568,17.8148],[0.0000,-0.3390,0.9408,0.0000],[-1,0,-1,0],[9E+09,0.0000,-635.3710,9E+09,9E+09,9E+09]];
	CONST robtarget p927:=[[0.0000,-163.9955,17.8344],[0.0000,-0.3346,0.9424,0.0000],[-1,0,-1,0],[9E+09,0.0000,-635.9061,9E+09,9E+09,9E+09]];
	CONST robtarget p928:=[[0.0000,-162.7488,17.8539],[0.0000,-0.3301,0.9439,0.0000],[-1,0,-1,0],[9E+09,0.0000,-636.4495,9E+09,9E+09,9E+09]];
	CONST robtarget p929:=[[0.0000,-161.5169,17.8734],[0.0000,-0.3256,0.9455,0.0000],[-1,0,-1,0],[9E+09,0.0000,-637.0013,9E+09,9E+09,9E+09]];
	CONST robtarget p930:=[[0.0000,-160.3002,17.8930],[0.0000,-0.3209,0.9471,0.0000],[-1,0,-1,0],[9E+09,0.0000,-637.5614,9E+09,9E+09,9E+09]];
	CONST robtarget p931:=[[0.0000,-159.0990,17.9125],[0.0000,-0.3162,0.9487,0.0000],[-1,0,-1,0],[9E+09,0.0000,-638.1301,9E+09,9E+09,9E+09]];
	CONST robtarget p932:=[[0.0000,-157.9138,17.9320],[0.0000,-0.3114,0.9503,0.0000],[-1,0,-1,0],[9E+09,0.0000,-638.7074,9E+09,9E+09,9E+09]];
	CONST robtarget p933:=[[0.0000,-156.7448,17.9516],[0.0000,-0.3066,0.9518,0.0000],[-1,0,-1,0],[9E+09,0.0000,-639.2933,9E+09,9E+09,9E+09]];
	CONST robtarget p934:=[[0.0000,-155.5925,17.9711],[0.0000,-0.3016,0.9534,0.0000],[-1,0,-1,0],[9E+09,0.0000,-639.8880,9E+09,9E+09,9E+09]];
	CONST robtarget p935:=[[0.0000,-154.4572,17.9906],[0.0000,-0.2966,0.9550,0.0000],[-1,0,-1,0],[9E+09,0.0000,-640.4915,9E+09,9E+09,9E+09]];
	CONST robtarget p936:=[[0.0000,-153.3393,18.0102],[0.0000,-0.2915,0.9566,0.0000],[-1,0,-1,0],[9E+09,0.0000,-641.1038,9E+09,9E+09,9E+09]];
	CONST robtarget p937:=[[0.0000,-152.2391,18.0297],[0.0000,-0.2863,0.9581,0.0000],[-1,0,-1,0],[9E+09,0.0000,-641.7251,9E+09,9E+09,9E+09]];
	CONST robtarget p938:=[[0.0000,-151.1572,18.0492],[0.0000,-0.2810,0.9597,0.0000],[-1,0,-1,0],[9E+09,0.0000,-642.3554,9E+09,9E+09,9E+09]];
	CONST robtarget p939:=[[0.0000,-150.0937,18.0688],[0.0000,-0.2757,0.9612,0.0000],[-1,0,-1,0],[9E+09,0.0000,-642.9946,9E+09,9E+09,9E+09]];
	CONST robtarget p940:=[[0.0000,-149.0492,18.0883],[0.0000,-0.2702,0.9628,0.0000],[-1,0,-1,0],[9E+09,0.0000,-643.6429,9E+09,9E+09,9E+09]];
	CONST robtarget p941:=[[0.0000,-148.0241,18.1078],[0.0000,-0.2647,0.9643,0.0000],[-1,0,-1,0],[9E+09,0.0000,-644.3003,9E+09,9E+09,9E+09]];
	CONST robtarget p942:=[[0.0000,-147.0187,18.1273],[0.0000,-0.2591,0.9659,0.0000],[-1,0,-1,0],[9E+09,0.0000,-644.9667,9E+09,9E+09,9E+09]];
	CONST robtarget p943:=[[0.0000,-146.0335,18.1469],[0.0000,-0.2534,0.9674,0.0000],[-1,0,-1,0],[9E+09,0.0000,-645.6422,9E+09,9E+09,9E+09]];
	CONST robtarget p944:=[[0.0000,-145.0688,18.1664],[0.0000,-0.2476,0.9689,0.0000],[-1,0,-1,0],[9E+09,0.0000,-646.3269,9E+09,9E+09,9E+09]];
	CONST robtarget p945:=[[0.0000,-144.1252,18.1859],[0.0000,-0.2417,0.9703,0.0000],[-1,0,-1,0],[9E+09,0.0000,-647.0205,9E+09,9E+09,9E+09]];
	CONST robtarget p946:=[[0.0000,-143.2029,18.2055],[0.0000,-0.2358,0.9718,0.0000],[-1,0,-1,0],[9E+09,0.0000,-647.7232,9E+09,9E+09,9E+09]];
	CONST robtarget p947:=[[0.0000,-142.3025,18.2250],[0.0000,-0.2298,0.9732,0.0000],[-1,0,-1,0],[9E+09,0.0000,-648.4349,9E+09,9E+09,9E+09]];
	CONST robtarget p948:=[[0.0000,-141.4243,18.2445],[0.0000,-0.2236,0.9747,0.0000],[-1,0,-1,0],[9E+09,0.0000,-649.1556,9E+09,9E+09,9E+09]];
	CONST robtarget p949:=[[0.0000,-140.5687,18.2641],[0.0000,-0.2174,0.9761,0.0000],[-1,0,-1,0],[9E+09,0.0000,-649.8852,9E+09,9E+09,9E+09]];
	CONST robtarget p950:=[[0.0000,-139.7363,18.2836],[0.0000,-0.2111,0.9775,0.0000],[-1,0,-1,0],[9E+09,0.0000,-650.6235,9E+09,9E+09,9E+09]];
	CONST robtarget p951:=[[0.0000,-138.9273,18.3031],[0.0000,-0.2047,0.9788,0.0000],[-1,0,-1,0],[9E+09,0.0000,-651.3706,9E+09,9E+09,9E+09]];
	CONST robtarget p952:=[[0.0000,-138.1421,18.3227],[0.0000,-0.1983,0.9801,0.0000],[-1,0,-1,0],[9E+09,0.0000,-652.1263,9E+09,9E+09,9E+09]];
	CONST robtarget p953:=[[0.0000,-137.3813,18.3422],[0.0000,-0.1917,0.9814,0.0000],[-1,0,-1,0],[9E+09,0.0000,-652.8906,9E+09,9E+09,9E+09]];
	CONST robtarget p954:=[[0.0000,-136.6452,18.3617],[0.0000,-0.1851,0.9827,0.0000],[-1,0,-1,0],[9E+09,0.0000,-653.6631,9E+09,9E+09,9E+09]];
	CONST robtarget p955:=[[0.0000,-135.9343,18.3813],[0.0000,-0.1784,0.9840,0.0000],[-1,0,-1,0],[9E+09,0.0000,-654.4440,9E+09,9E+09,9E+09]];
	CONST robtarget p956:=[[0.0000,-135.2488,18.4008],[0.0000,-0.1716,0.9852,0.0000],[-1,0,-1,0],[9E+09,0.0000,-655.2328,9E+09,9E+09,9E+09]];
	CONST robtarget p957:=[[0.0000,-134.5892,18.4203],[0.0000,-0.1648,0.9863,0.0000],[-1,0,-1,0],[9E+09,0.0000,-656.0296,9E+09,9E+09,9E+09]];
	CONST robtarget p958:=[[0.0000,-133.9559,18.4398],[0.0000,-0.1579,0.9875,0.0000],[-1,0,-1,0],[9E+09,0.0000,-656.8340,9E+09,9E+09,9E+09]];
	CONST robtarget p959:=[[0.0000,-133.3493,18.4594],[0.0000,-0.1509,0.9886,0.0000],[-1,0,-1,0],[9E+09,0.0000,-657.6460,9E+09,9E+09,9E+09]];
	CONST robtarget p960:=[[0.0000,-132.7697,18.4789],[0.0000,-0.1438,0.9896,0.0000],[-1,0,-1,0],[9E+09,0.0000,-658.4652,9E+09,9E+09,9E+09]];
	CONST robtarget p961:=[[0.0000,-132.2174,18.4984],[0.0000,-0.1367,0.9906,0.0000],[-1,0,-1,0],[9E+09,0.0000,-659.2914,9E+09,9E+09,9E+09]];
	CONST robtarget p962:=[[0.0000,-131.6929,18.5180],[0.0000,-0.1295,0.9916,0.0000],[-1,0,-1,0],[9E+09,0.0000,-660.1243,9E+09,9E+09,9E+09]];
	CONST robtarget p963:=[[0.0000,-131.1964,18.5375],[0.0000,-0.1222,0.9925,0.0000],[-1,0,-1,0],[9E+09,0.0000,-660.9638,9E+09,9E+09,9E+09]];
	CONST robtarget p964:=[[0.0000,-130.7283,18.5570],[0.0000,-0.1149,0.9934,0.0000],[-1,0,-1,0],[9E+09,0.0000,-661.8094,9E+09,9E+09,9E+09]];
	CONST robtarget p965:=[[0.0000,-130.2889,18.5766],[0.0000,-0.1075,0.9942,0.0000],[-1,0,-1,0],[9E+09,0.0000,-662.6609,9E+09,9E+09,9E+09]];
	CONST robtarget p966:=[[0.0000,-129.8784,18.5961],[0.0000,-0.1000,0.9950,0.0000],[-1,0,-1,0],[9E+09,0.0000,-663.5180,9E+09,9E+09,9E+09]];
	CONST robtarget p967:=[[0.0000,-129.4972,18.6156],[0.0000,-0.0925,0.9957,0.0000],[-1,0,-1,0],[9E+09,0.0000,-664.3803,9E+09,9E+09,9E+09]];
	CONST robtarget p968:=[[0.0000,-129.1455,18.6352],[0.0000,-0.0850,0.9964,0.0000],[-1,0,-1,0],[9E+09,0.0000,-665.2476,9E+09,9E+09,9E+09]];
	CONST robtarget p969:=[[0.0000,-128.8236,18.6547],[0.0000,-0.0774,0.9970,0.0000],[-1,0,-1,0],[9E+09,0.0000,-666.1193,9E+09,9E+09,9E+09]];
	CONST robtarget p970:=[[0.0000,-128.5316,18.6742],[0.0000,-0.0698,0.9976,0.0000],[-1,0,-1,0],[9E+09,0.0000,-666.9953,9E+09,9E+09,9E+09]];
	CONST robtarget p971:=[[0.0000,-128.2697,18.6938],[0.0000,-0.0621,0.9981,0.0000],[-1,0,-1,0],[9E+09,0.0000,-667.8750,9E+09,9E+09,9E+09]];
	CONST robtarget p972:=[[0.0000,-128.0383,18.7133],[0.0000,-0.0544,0.9985,0.0000],[-1,0,-1,0],[9E+09,0.0000,-668.7581,9E+09,9E+09,9E+09]];
	CONST robtarget p973:=[[0.0000,-127.8373,18.7328],[0.0000,-0.0467,0.9989,0.0000],[-1,0,-1,0],[9E+09,0.0000,-669.6442,9E+09,9E+09,9E+09]];
	CONST robtarget p974:=[[0.0000,-127.6671,18.7523],[0.0000,-0.0390,0.9992,0.0000],[-1,0,-1,0],[9E+09,0.0000,-670.5328,9E+09,9E+09,9E+09]];
	CONST robtarget p975:=[[0.0000,-127.5276,18.7719],[0.0000,-0.0312,0.9995,0.0000],[-1,0,-1,0],[9E+09,0.0000,-671.4237,9E+09,9E+09,9E+09]];
	CONST robtarget p976:=[[0.0000,-127.4190,18.7914],[0.0000,-0.0234,0.9997,0.0000],[-1,0,-1,0],[9E+09,0.0000,-672.3162,9E+09,9E+09,9E+09]];
	CONST robtarget p977:=[[0.0000,-127.3414,18.8109],[0.0000,-0.0156,0.9999,0.0000],[-1,0,-1,0],[9E+09,0.0000,-673.2101,9E+09,9E+09,9E+09]];
	CONST robtarget p978:=[[0.0000,-127.2948,18.8305],[0.0000,-0.0078,1.0000,0.0000],[-1,0,-1,0],[9E+09,0.0000,-674.1048,9E+09,9E+09,9E+09]];
	CONST robtarget p979:=[[0.0000,-127.2792,18.8500],[0.0000,0.0000,1.0000,0.0000],[-1,0,-1,0],[9E+09,0.0000,-675.0000,9E+09,9E+09,9E+09]];
	CONST robtarget p980:=[[0.0000,-127.2948,18.8695],[0.0000,-0.0078,-1.0000,0.0000],[-1,0,-1,0],[9E+09,0.0000,-675.8952,9E+09,9E+09,9E+09]];
	CONST robtarget p981:=[[0.0000,-127.3414,18.8891],[0.0000,-0.0156,-0.9999,0.0000],[-1,0,-1,0],[9E+09,0.0000,-676.7899,9E+09,9E+09,9E+09]];
	CONST robtarget p982:=[[0.0000,-127.4190,18.9086],[0.0000,-0.0234,-0.9997,0.0000],[-1,0,-1,0],[9E+09,0.0000,-677.6838,9E+09,9E+09,9E+09]];
	CONST robtarget p983:=[[0.0000,-127.5276,18.9281],[0.0000,-0.0312,-0.9995,0.0000],[-1,0,-1,0],[9E+09,0.0000,-678.5763,9E+09,9E+09,9E+09]];
	CONST robtarget p984:=[[0.0000,-127.6671,18.9477],[0.0000,-0.0390,-0.9992,0.0000],[-1,0,-1,0],[9E+09,0.0000,-679.4672,9E+09,9E+09,9E+09]];
	CONST robtarget p985:=[[0.0000,-127.8373,18.9672],[0.0000,-0.0467,-0.9989,0.0000],[-1,0,-1,0],[9E+09,0.0000,-680.3558,9E+09,9E+09,9E+09]];
	CONST robtarget p986:=[[0.0000,-128.0383,18.9867],[0.0000,-0.0544,-0.9985,0.0000],[-1,0,-1,0],[9E+09,0.0000,-681.2419,9E+09,9E+09,9E+09]];
	CONST robtarget p987:=[[0.0000,-128.2697,19.0063],[0.0000,-0.0621,-0.9981,0.0000],[-1,0,-1,0],[9E+09,0.0000,-682.1250,9E+09,9E+09,9E+09]];
	CONST robtarget p988:=[[0.0000,-128.5316,19.0258],[0.0000,-0.0698,-0.9976,0.0000],[-1,0,-1,0],[9E+09,0.0000,-683.0047,9E+09,9E+09,9E+09]];
	CONST robtarget p989:=[[0.0000,-128.8236,19.0453],[0.0000,-0.0774,-0.9970,0.0000],[-1,0,-1,0],[9E+09,0.0000,-683.8807,9E+09,9E+09,9E+09]];
	CONST robtarget p990:=[[0.0000,-129.1455,19.0648],[0.0000,-0.0850,-0.9964,0.0000],[-1,0,-1,0],[9E+09,0.0000,-684.7524,9E+09,9E+09,9E+09]];
	CONST robtarget p991:=[[0.0000,-129.4972,19.0844],[0.0000,-0.0925,-0.9957,0.0000],[-1,0,-1,0],[9E+09,0.0000,-685.6197,9E+09,9E+09,9E+09]];
	CONST robtarget p992:=[[0.0000,-129.8784,19.1039],[0.0000,-0.1000,-0.9950,0.0000],[-1,0,-1,0],[9E+09,0.0000,-686.4820,9E+09,9E+09,9E+09]];
	CONST robtarget p993:=[[0.0000,-130.2889,19.1234],[0.0000,-0.1075,-0.9942,0.0000],[-1,0,-1,0],[9E+09,0.0000,-687.3391,9E+09,9E+09,9E+09]];
	CONST robtarget p994:=[[0.0000,-130.7283,19.1430],[0.0000,-0.1149,-0.9934,0.0000],[-1,0,-1,0],[9E+09,0.0000,-688.1906,9E+09,9E+09,9E+09]];
	CONST robtarget p995:=[[0.0000,-131.1964,19.1625],[0.0000,-0.1222,-0.9925,0.0000],[-1,0,-1,0],[9E+09,0.0000,-689.0362,9E+09,9E+09,9E+09]];
	CONST robtarget p996:=[[0.0000,-131.6929,19.1820],[0.0000,-0.1295,-0.9916,0.0000],[-1,0,-1,0],[9E+09,0.0000,-689.8757,9E+09,9E+09,9E+09]];
	CONST robtarget p997:=[[0.0000,-132.2174,19.2016],[0.0000,-0.1367,-0.9906,0.0000],[-1,0,-1,0],[9E+09,0.0000,-690.7086,9E+09,9E+09,9E+09]];
	CONST robtarget p998:=[[0.0000,-132.7697,19.2211],[0.0000,-0.1438,-0.9896,0.0000],[-1,0,-1,0],[9E+09,0.0000,-691.5348,9E+09,9E+09,9E+09]];
	CONST robtarget p999:=[[0.0000,-133.3493,19.2406],[0.0000,-0.1509,-0.9886,0.0000],[-1,0,-1,0],[9E+09,0.0000,-692.3540,9E+09,9E+09,9E+09]];
	VAR speeddata vd1 :=[50.00,500,5000,50.00];
	VAR speeddata vd2 :=[7.23,500,5000,2.04];
	VAR speeddata vd3 :=[7.18,500,5000,2.07];
	VAR speeddata vd4 :=[7.13,500,5000,2.10];
	VAR speeddata vd5 :=[7.08,500,5000,2.13];
	VAR speeddata vd6 :=[7.03,500,5000,2.16];
	VAR speeddata vd7 :=[6.97,500,5000,2.19];
	VAR speeddata vd8 :=[6.92,500,5000,2.23];
	VAR speeddata vd9 :=[6.86,500,5000,2.26];
	VAR speeddata vd10 :=[6.80,500,5000,2.29];
	VAR speeddata vd11 :=[6.74,500,5000,2.33];
	VAR speeddata vd12 :=[6.68,500,5000,2.36];
	VAR speeddata vd13 :=[6.62,500,5000,2.40];
	VAR speeddata vd14 :=[6.56,500,5000,2.43];
	VAR speeddata vd15 :=[6.49,500,5000,2.47];
	VAR speeddata vd16 :=[6.43,500,5000,2.51];
	VAR speeddata vd17 :=[6.36,500,5000,2.54];
	VAR speeddata vd18 :=[6.29,500,5000,2.58];
	VAR speeddata vd19 :=[6.22,500,5000,2.62];
	VAR speeddata vd20 :=[6.15,500,5000,2.66];
	VAR speeddata vd21 :=[6.07,500,5000,2.69];
	VAR speeddata vd22 :=[6.00,500,5000,2.73];
	VAR speeddata vd23 :=[5.92,500,5000,2.77];
	VAR speeddata vd24 :=[5.84,500,5000,2.81];
	VAR speeddata vd25 :=[5.76,500,5000,2.85];
	VAR speeddata vd26 :=[5.68,500,5000,2.89];
	VAR speeddata vd27 :=[5.60,500,5000,2.93];
	VAR speeddata vd28 :=[5.51,500,5000,2.97];
	VAR speeddata vd29 :=[5.43,500,5000,3.01];
	VAR speeddata vd30 :=[5.34,500,5000,3.05];
	VAR speeddata vd31 :=[5.25,500,5000,3.09];
	VAR speeddata vd32 :=[5.15,500,5000,3.14];
	VAR speeddata vd33 :=[5.06,500,5000,3.18];
	VAR speeddata vd34 :=[4.96,500,5000,3.22];
	VAR speeddata vd35 :=[4.87,500,5000,3.26];
	VAR speeddata vd36 :=[4.77,500,5000,3.30];
	VAR speeddata vd37 :=[4.66,500,5000,3.34];
	VAR speeddata vd38 :=[4.56,500,5000,3.38];
	VAR speeddata vd39 :=[4.45,500,5000,3.42];
	VAR speeddata vd40 :=[4.35,500,5000,3.46];
	VAR speeddata vd41 :=[4.24,500,5000,3.50];
	VAR speeddata vd42 :=[4.13,500,5000,3.54];
	VAR speeddata vd43 :=[4.01,500,5000,3.58];
	VAR speeddata vd44 :=[3.90,500,5000,3.62];
	VAR speeddata vd45 :=[3.78,500,5000,3.66];
	VAR speeddata vd46 :=[3.66,500,5000,3.70];
	VAR speeddata vd47 :=[3.54,500,5000,3.73];
	VAR speeddata vd48 :=[3.42,500,5000,3.77];
	VAR speeddata vd49 :=[3.30,500,5000,3.81];
	VAR speeddata vd50 :=[3.17,500,5000,3.84];
	VAR speeddata vd51 :=[3.04,500,5000,3.87];
	VAR speeddata vd52 :=[2.92,500,5000,3.91];
	VAR speeddata vd53 :=[2.78,500,5000,3.94];
	VAR speeddata vd54 :=[2.65,500,5000,3.97];
	VAR speeddata vd55 :=[2.52,500,5000,4.00];
	VAR speeddata vd56 :=[2.38,500,5000,4.03];
	VAR speeddata vd57 :=[2.25,500,5000,4.05];
	VAR speeddata vd58 :=[2.11,500,5000,4.08];
	VAR speeddata vd59 :=[1.97,500,5000,4.10];
	VAR speeddata vd60 :=[1.83,500,5000,4.13];
	VAR speeddata vd61 :=[1.69,500,5000,4.15];
	VAR speeddata vd62 :=[1.55,500,5000,4.17];
	VAR speeddata vd63 :=[1.40,500,5000,4.19];
	VAR speeddata vd64 :=[1.26,500,5000,4.20];
	VAR speeddata vd65 :=[1.11,500,5000,4.22];
	VAR speeddata vd66 :=[0.97,500,5000,4.23];
	VAR speeddata vd67 :=[0.82,500,5000,4.24];
	VAR speeddata vd68 :=[0.68,500,5000,4.25];
	VAR speeddata vd69 :=[0.53,500,5000,4.26];
	VAR speeddata vd70 :=[0.39,500,5000,4.26];
	VAR speeddata vd71 :=[0.25,500,5000,4.27];
	VAR speeddata vd72 :=[0.12,500,5000,4.27];
	VAR speeddata vd73 :=[0.12,500,5000,4.27];
	VAR speeddata vd74 :=[0.24,500,5000,4.27];
	VAR speeddata vd75 :=[0.38,500,5000,4.26];
	VAR speeddata vd76 :=[0.52,500,5000,4.26];
	VAR speeddata vd77 :=[0.67,500,5000,4.25];
	VAR speeddata vd78 :=[0.81,500,5000,4.24];
	VAR speeddata vd79 :=[0.96,500,5000,4.23];
	VAR speeddata vd80 :=[1.10,500,5000,4.22];
	VAR speeddata vd81 :=[1.25,500,5000,4.20];
	VAR speeddata vd82 :=[1.39,500,5000,4.19];
	VAR speeddata vd83 :=[1.54,500,5000,4.17];
	VAR speeddata vd84 :=[1.68,500,5000,4.15];
	VAR speeddata vd85 :=[1.82,500,5000,4.13];
	VAR speeddata vd86 :=[1.96,500,5000,4.11];
	VAR speeddata vd87 :=[2.10,500,5000,4.08];
	VAR speeddata vd88 :=[2.24,500,5000,4.06];
	VAR speeddata vd89 :=[2.37,500,5000,4.03];
	VAR speeddata vd90 :=[2.51,500,5000,4.00];
	VAR speeddata vd91 :=[2.64,500,5000,3.97];
	VAR speeddata vd92 :=[2.78,500,5000,3.94];
	VAR speeddata vd93 :=[2.91,500,5000,3.91];
	VAR speeddata vd94 :=[3.04,500,5000,3.88];
	VAR speeddata vd95 :=[3.16,500,5000,3.84];
	VAR speeddata vd96 :=[3.29,500,5000,3.81];
	VAR speeddata vd97 :=[3.41,500,5000,3.77];
	VAR speeddata vd98 :=[3.54,500,5000,3.74];
	VAR speeddata vd99 :=[3.66,500,5000,3.70];
	VAR speeddata vd100 :=[3.77,500,5000,3.66];
	VAR speeddata vd101 :=[3.89,500,5000,3.62];
	VAR speeddata vd102 :=[4.01,500,5000,3.58];
	VAR speeddata vd103 :=[4.12,500,5000,3.55];
	VAR speeddata vd104 :=[4.23,500,5000,3.51];
	VAR speeddata vd105 :=[4.34,500,5000,3.47];
	VAR speeddata vd106 :=[4.45,500,5000,3.43];
	VAR speeddata vd107 :=[4.55,500,5000,3.38];
	VAR speeddata vd108 :=[4.66,500,5000,3.34];
	VAR speeddata vd109 :=[4.76,500,5000,3.30];
	VAR speeddata vd110 :=[4.86,500,5000,3.26];
	VAR speeddata vd111 :=[4.96,500,5000,3.22];
	VAR speeddata vd112 :=[5.05,500,5000,3.18];
	VAR speeddata vd113 :=[5.15,500,5000,3.14];
	VAR speeddata vd114 :=[5.24,500,5000,3.10];
	VAR speeddata vd115 :=[5.33,500,5000,3.06];
	VAR speeddata vd116 :=[5.42,500,5000,3.02];
	VAR speeddata vd117 :=[5.51,500,5000,2.97];
	VAR speeddata vd118 :=[5.59,500,5000,2.93];
	VAR speeddata vd119 :=[5.68,500,5000,2.89];
	VAR speeddata vd120 :=[5.76,500,5000,2.85];
	VAR speeddata vd121 :=[5.84,500,5000,2.81];
	VAR speeddata vd122 :=[5.92,500,5000,2.77];
	VAR speeddata vd123 :=[5.99,500,5000,2.74];
	VAR speeddata vd124 :=[6.07,500,5000,2.70];
	VAR speeddata vd125 :=[6.14,500,5000,2.66];
	VAR speeddata vd126 :=[6.21,500,5000,2.62];
	VAR speeddata vd127 :=[6.29,500,5000,2.58];
	VAR speeddata vd128 :=[6.35,500,5000,2.55];
	VAR speeddata vd129 :=[6.42,500,5000,2.51];
	VAR speeddata vd130 :=[6.49,500,5000,2.47];
	VAR speeddata vd131 :=[6.55,500,5000,2.44];
	VAR speeddata vd132 :=[6.62,500,5000,2.40];
	VAR speeddata vd133 :=[6.68,500,5000,2.37];
	VAR speeddata vd134 :=[6.74,500,5000,2.33];
	VAR speeddata vd135 :=[6.80,500,5000,2.30];
	VAR speeddata vd136 :=[6.86,500,5000,2.26];
	VAR speeddata vd137 :=[7.04,500,5000,2.21];
	VAR speeddata vd138 :=[6.99,500,5000,2.24];
	VAR speeddata vd139 :=[6.93,500,5000,2.28];
	VAR speeddata vd140 :=[6.87,500,5000,2.31];
	VAR speeddata vd141 :=[6.82,500,5000,2.35];
	VAR speeddata vd142 :=[6.76,500,5000,2.38];
	VAR speeddata vd143 :=[6.69,500,5000,2.42];
	VAR speeddata vd144 :=[6.63,500,5000,2.45];
	VAR speeddata vd145 :=[6.56,500,5000,2.49];
	VAR speeddata vd146 :=[6.50,500,5000,2.53];
	VAR speeddata vd147 :=[6.43,500,5000,2.57];
	VAR speeddata vd148 :=[6.36,500,5000,2.61];
	VAR speeddata vd149 :=[6.29,500,5000,2.65];
	VAR speeddata vd150 :=[6.22,500,5000,2.69];
	VAR speeddata vd151 :=[6.14,500,5000,2.73];
	VAR speeddata vd152 :=[6.07,500,5000,2.77];
	VAR speeddata vd153 :=[5.99,500,5000,2.81];
	VAR speeddata vd154 :=[5.91,500,5000,2.85];
	VAR speeddata vd155 :=[5.83,500,5000,2.89];
	VAR speeddata vd156 :=[5.75,500,5000,2.93];
	VAR speeddata vd157 :=[5.66,500,5000,2.98];
	VAR speeddata vd158 :=[5.58,500,5000,3.02];
	VAR speeddata vd159 :=[5.49,500,5000,3.06];
	VAR speeddata vd160 :=[5.40,500,5000,3.10];
	VAR speeddata vd161 :=[5.31,500,5000,3.15];
	VAR speeddata vd162 :=[5.21,500,5000,3.19];
	VAR speeddata vd163 :=[5.12,500,5000,3.23];
	VAR speeddata vd164 :=[5.02,500,5000,3.28];
	VAR speeddata vd165 :=[4.92,500,5000,3.32];
	VAR speeddata vd166 :=[4.82,500,5000,3.36];
	VAR speeddata vd167 :=[4.71,500,5000,3.41];
	VAR speeddata vd168 :=[4.61,500,5000,3.45];
	VAR speeddata vd169 :=[4.50,500,5000,3.49];
	VAR speeddata vd170 :=[4.39,500,5000,3.54];
	VAR speeddata vd171 :=[4.28,500,5000,3.58];
	VAR speeddata vd172 :=[4.16,500,5000,3.62];
	VAR speeddata vd173 :=[4.05,500,5000,3.66];
	VAR speeddata vd174 :=[3.93,500,5000,3.70];
	VAR speeddata vd175 :=[3.81,500,5000,3.74];
	VAR speeddata vd176 :=[3.69,500,5000,3.78];
	VAR speeddata vd177 :=[3.57,500,5000,3.82];
	VAR speeddata vd178 :=[3.44,500,5000,3.86];
	VAR speeddata vd179 :=[3.31,500,5000,3.90];
	VAR speeddata vd180 :=[3.19,500,5000,3.94];
	VAR speeddata vd181 :=[3.05,500,5000,3.97];
	VAR speeddata vd182 :=[2.92,500,5000,4.01];
	VAR speeddata vd183 :=[2.79,500,5000,4.04];
	VAR speeddata vd184 :=[2.65,500,5000,4.07];
	VAR speeddata vd185 :=[2.51,500,5000,4.10];
	VAR speeddata vd186 :=[2.37,500,5000,4.13];
	VAR speeddata vd187 :=[2.23,500,5000,4.16];
	VAR speeddata vd188 :=[2.09,500,5000,4.19];
	VAR speeddata vd189 :=[1.95,500,5000,4.21];
	VAR speeddata vd190 :=[1.80,500,5000,4.24];
	VAR speeddata vd191 :=[1.66,500,5000,4.26];
	VAR speeddata vd192 :=[1.51,500,5000,4.28];
	VAR speeddata vd193 :=[1.36,500,5000,4.30];
	VAR speeddata vd194 :=[1.22,500,5000,4.32];
	VAR speeddata vd195 :=[1.07,500,5000,4.33];
	VAR speeddata vd196 :=[0.92,500,5000,4.34];
	VAR speeddata vd197 :=[0.77,500,5000,4.35];
	VAR speeddata vd198 :=[0.62,500,5000,4.36];
	VAR speeddata vd199 :=[0.47,500,5000,4.37];
	VAR speeddata vd200 :=[0.32,500,5000,4.38];
	VAR speeddata vd201 :=[0.18,500,5000,4.38];
	VAR speeddata vd202 :=[0.10,500,5000,4.38];
	VAR speeddata vd203 :=[0.18,500,5000,4.38];
	VAR speeddata vd204 :=[0.32,500,5000,4.38];
	VAR speeddata vd205 :=[0.47,500,5000,4.37];
	VAR speeddata vd206 :=[0.62,500,5000,4.36];
	VAR speeddata vd207 :=[0.77,500,5000,4.35];
	VAR speeddata vd208 :=[0.92,500,5000,4.34];
	VAR speeddata vd209 :=[1.07,500,5000,4.33];
	VAR speeddata vd210 :=[1.22,500,5000,4.32];
	VAR speeddata vd211 :=[1.36,500,5000,4.30];
	VAR speeddata vd212 :=[1.51,500,5000,4.28];
	VAR speeddata vd213 :=[1.66,500,5000,4.26];
	VAR speeddata vd214 :=[1.80,500,5000,4.24];
	VAR speeddata vd215 :=[1.95,500,5000,4.21];
	VAR speeddata vd216 :=[2.09,500,5000,4.19];
	VAR speeddata vd217 :=[2.23,500,5000,4.16];
	VAR speeddata vd218 :=[2.37,500,5000,4.13];
	VAR speeddata vd219 :=[2.51,500,5000,4.10];
	VAR speeddata vd220 :=[2.65,500,5000,4.07];
	VAR speeddata vd221 :=[2.79,500,5000,4.04];
	VAR speeddata vd222 :=[2.92,500,5000,4.01];
	VAR speeddata vd223 :=[3.05,500,5000,3.97];
	VAR speeddata vd224 :=[3.19,500,5000,3.94];
	VAR speeddata vd225 :=[3.31,500,5000,3.90];
	VAR speeddata vd226 :=[3.44,500,5000,3.86];
	VAR speeddata vd227 :=[3.57,500,5000,3.82];
	VAR speeddata vd228 :=[3.69,500,5000,3.78];
	VAR speeddata vd229 :=[3.81,500,5000,3.74];
	VAR speeddata vd230 :=[3.93,500,5000,3.70];
	VAR speeddata vd231 :=[4.05,500,5000,3.66];
	VAR speeddata vd232 :=[4.16,500,5000,3.62];
	VAR speeddata vd233 :=[4.28,500,5000,3.58];
	VAR speeddata vd234 :=[4.39,500,5000,3.54];
	VAR speeddata vd235 :=[4.50,500,5000,3.49];
	VAR speeddata vd236 :=[4.61,500,5000,3.45];
	VAR speeddata vd237 :=[4.71,500,5000,3.41];
	VAR speeddata vd238 :=[4.82,500,5000,3.36];
	VAR speeddata vd239 :=[4.92,500,5000,3.32];
	VAR speeddata vd240 :=[5.02,500,5000,3.28];
	VAR speeddata vd241 :=[5.12,500,5000,3.23];
	VAR speeddata vd242 :=[5.21,500,5000,3.19];
	VAR speeddata vd243 :=[5.31,500,5000,3.15];
	VAR speeddata vd244 :=[5.40,500,5000,3.10];
	VAR speeddata vd245 :=[5.49,500,5000,3.06];
	VAR speeddata vd246 :=[5.58,500,5000,3.02];
	VAR speeddata vd247 :=[5.66,500,5000,2.98];
	VAR speeddata vd248 :=[5.75,500,5000,2.93];
	VAR speeddata vd249 :=[5.83,500,5000,2.89];
	VAR speeddata vd250 :=[5.91,500,5000,2.85];
	VAR speeddata vd251 :=[5.99,500,5000,2.81];
	VAR speeddata vd252 :=[6.07,500,5000,2.77];
	VAR speeddata vd253 :=[6.14,500,5000,2.73];
	VAR speeddata vd254 :=[6.22,500,5000,2.69];
	VAR speeddata vd255 :=[6.29,500,5000,2.65];
	VAR speeddata vd256 :=[6.36,500,5000,2.61];
	VAR speeddata vd257 :=[6.43,500,5000,2.57];
	VAR speeddata vd258 :=[6.50,500,5000,2.53];
	VAR speeddata vd259 :=[6.56,500,5000,2.49];
	VAR speeddata vd260 :=[6.63,500,5000,2.45];
	VAR speeddata vd261 :=[6.69,500,5000,2.42];
	VAR speeddata vd262 :=[6.76,500,5000,2.38];
	VAR speeddata vd263 :=[6.82,500,5000,2.35];
	VAR speeddata vd264 :=[6.87,500,5000,2.31];
	VAR speeddata vd265 :=[6.93,500,5000,2.28];
	VAR speeddata vd266 :=[6.99,500,5000,2.24];
	VAR speeddata vd267 :=[7.04,500,5000,2.21];
	VAR speeddata vd268 :=[7.04,500,5000,2.21];
	VAR speeddata vd269 :=[6.99,500,5000,2.24];
	VAR speeddata vd270 :=[6.93,500,5000,2.28];
	VAR speeddata vd271 :=[6.87,500,5000,2.31];
	VAR speeddata vd272 :=[6.82,500,5000,2.35];
	VAR speeddata vd273 :=[6.76,500,5000,2.38];
	VAR speeddata vd274 :=[6.69,500,5000,2.42];
	VAR speeddata vd275 :=[6.63,500,5000,2.45];
	VAR speeddata vd276 :=[6.56,500,5000,2.49];
	VAR speeddata vd277 :=[6.50,500,5000,2.53];
	VAR speeddata vd278 :=[6.43,500,5000,2.57];
	VAR speeddata vd279 :=[6.36,500,5000,2.61];
	VAR speeddata vd280 :=[6.29,500,5000,2.65];
	VAR speeddata vd281 :=[6.22,500,5000,2.69];
	VAR speeddata vd282 :=[6.14,500,5000,2.73];
	VAR speeddata vd283 :=[6.07,500,5000,2.77];
	VAR speeddata vd284 :=[5.99,500,5000,2.81];
	VAR speeddata vd285 :=[5.91,500,5000,2.85];
	VAR speeddata vd286 :=[5.83,500,5000,2.89];
	VAR speeddata vd287 :=[5.75,500,5000,2.93];
	VAR speeddata vd288 :=[5.66,500,5000,2.98];
	VAR speeddata vd289 :=[5.58,500,5000,3.02];
	VAR speeddata vd290 :=[5.49,500,5000,3.06];
	VAR speeddata vd291 :=[5.40,500,5000,3.10];
	VAR speeddata vd292 :=[5.31,500,5000,3.15];
	VAR speeddata vd293 :=[5.21,500,5000,3.19];
	VAR speeddata vd294 :=[5.12,500,5000,3.23];
	VAR speeddata vd295 :=[5.02,500,5000,3.28];
	VAR speeddata vd296 :=[4.92,500,5000,3.32];
	VAR speeddata vd297 :=[4.82,500,5000,3.36];
	VAR speeddata vd298 :=[4.71,500,5000,3.41];
	VAR speeddata vd299 :=[4.61,500,5000,3.45];
	VAR speeddata vd300 :=[4.50,500,5000,3.49];
	VAR speeddata vd301 :=[4.39,500,5000,3.54];
	VAR speeddata vd302 :=[4.28,500,5000,3.58];
	VAR speeddata vd303 :=[4.16,500,5000,3.62];
	VAR speeddata vd304 :=[4.05,500,5000,3.66];
	VAR speeddata vd305 :=[3.93,500,5000,3.70];
	VAR speeddata vd306 :=[3.81,500,5000,3.74];
	VAR speeddata vd307 :=[3.69,500,5000,3.78];
	VAR speeddata vd308 :=[3.57,500,5000,3.82];
	VAR speeddata vd309 :=[3.44,500,5000,3.86];
	VAR speeddata vd310 :=[3.31,500,5000,3.90];
	VAR speeddata vd311 :=[3.19,500,5000,3.94];
	VAR speeddata vd312 :=[3.05,500,5000,3.97];
	VAR speeddata vd313 :=[2.92,500,5000,4.01];
	VAR speeddata vd314 :=[2.79,500,5000,4.04];
	VAR speeddata vd315 :=[2.65,500,5000,4.07];
	VAR speeddata vd316 :=[2.51,500,5000,4.10];
	VAR speeddata vd317 :=[2.37,500,5000,4.13];
	VAR speeddata vd318 :=[2.23,500,5000,4.16];
	VAR speeddata vd319 :=[2.09,500,5000,4.19];
	VAR speeddata vd320 :=[1.95,500,5000,4.21];
	VAR speeddata vd321 :=[1.80,500,5000,4.24];
	VAR speeddata vd322 :=[1.66,500,5000,4.26];
	VAR speeddata vd323 :=[1.51,500,5000,4.28];
	VAR speeddata vd324 :=[1.36,500,5000,4.30];
	VAR speeddata vd325 :=[1.22,500,5000,4.32];
	VAR speeddata vd326 :=[1.07,500,5000,4.33];
	VAR speeddata vd327 :=[0.92,500,5000,4.34];
	VAR speeddata vd328 :=[0.77,500,5000,4.35];
	VAR speeddata vd329 :=[0.62,500,5000,4.36];
	VAR speeddata vd330 :=[0.47,500,5000,4.37];
	VAR speeddata vd331 :=[0.32,500,5000,4.38];
	VAR speeddata vd332 :=[0.18,500,5000,4.38];
	VAR speeddata vd333 :=[0.10,500,5000,4.38];
	VAR speeddata vd334 :=[0.18,500,5000,4.38];
	VAR speeddata vd335 :=[0.32,500,5000,4.38];
	VAR speeddata vd336 :=[0.47,500,5000,4.37];
	VAR speeddata vd337 :=[0.62,500,5000,4.36];
	VAR speeddata vd338 :=[0.77,500,5000,4.35];
	VAR speeddata vd339 :=[0.92,500,5000,4.34];
	VAR speeddata vd340 :=[1.07,500,5000,4.33];
	VAR speeddata vd341 :=[1.22,500,5000,4.32];
	VAR speeddata vd342 :=[1.36,500,5000,4.30];
	VAR speeddata vd343 :=[1.51,500,5000,4.28];
	VAR speeddata vd344 :=[1.66,500,5000,4.26];
	VAR speeddata vd345 :=[1.80,500,5000,4.24];
	VAR speeddata vd346 :=[1.95,500,5000,4.21];
	VAR speeddata vd347 :=[2.09,500,5000,4.19];
	VAR speeddata vd348 :=[2.23,500,5000,4.16];
	VAR speeddata vd349 :=[2.37,500,5000,4.13];
	VAR speeddata vd350 :=[2.51,500,5000,4.10];
	VAR speeddata vd351 :=[2.65,500,5000,4.07];
	VAR speeddata vd352 :=[2.79,500,5000,4.04];
	VAR speeddata vd353 :=[2.92,500,5000,4.01];
	VAR speeddata vd354 :=[3.05,500,5000,3.97];
	VAR speeddata vd355 :=[3.19,500,5000,3.94];
	VAR speeddata vd356 :=[3.31,500,5000,3.90];
	VAR speeddata vd357 :=[3.44,500,5000,3.86];
	VAR speeddata vd358 :=[3.57,500,5000,3.82];
	VAR speeddata vd359 :=[3.69,500,5000,3.78];
	VAR speeddata vd360 :=[3.81,500,5000,3.74];
	VAR speeddata vd361 :=[3.93,500,5000,3.70];
	VAR speeddata vd362 :=[4.05,500,5000,3.66];
	VAR speeddata vd363 :=[4.16,500,5000,3.62];
	VAR speeddata vd364 :=[4.28,500,5000,3.58];
	VAR speeddata vd365 :=[4.39,500,5000,3.54];
	VAR speeddata vd366 :=[4.50,500,5000,3.49];
	VAR speeddata vd367 :=[4.61,500,5000,3.45];
	VAR speeddata vd368 :=[4.71,500,5000,3.41];
	VAR speeddata vd369 :=[4.82,500,5000,3.36];
	VAR speeddata vd370 :=[4.92,500,5000,3.32];
	VAR speeddata vd371 :=[5.02,500,5000,3.28];
	VAR speeddata vd372 :=[5.12,500,5000,3.23];
	VAR speeddata vd373 :=[5.21,500,5000,3.19];
	VAR speeddata vd374 :=[5.31,500,5000,3.15];
	VAR speeddata vd375 :=[5.40,500,5000,3.10];
	VAR speeddata vd376 :=[5.49,500,5000,3.06];
	VAR speeddata vd377 :=[5.58,500,5000,3.02];
	VAR speeddata vd378 :=[5.66,500,5000,2.98];
	VAR speeddata vd379 :=[5.75,500,5000,2.93];
	VAR speeddata vd380 :=[5.83,500,5000,2.89];
	VAR speeddata vd381 :=[5.91,500,5000,2.85];
	VAR speeddata vd382 :=[5.99,500,5000,2.81];
	VAR speeddata vd383 :=[6.07,500,5000,2.77];
	VAR speeddata vd384 :=[6.14,500,5000,2.73];
	VAR speeddata vd385 :=[6.22,500,5000,2.69];
	VAR speeddata vd386 :=[6.29,500,5000,2.65];
	VAR speeddata vd387 :=[6.36,500,5000,2.61];
	VAR speeddata vd388 :=[6.43,500,5000,2.57];
	VAR speeddata vd389 :=[6.50,500,5000,2.53];
	VAR speeddata vd390 :=[6.56,500,5000,2.49];
	VAR speeddata vd391 :=[6.63,500,5000,2.45];
	VAR speeddata vd392 :=[6.69,500,5000,2.42];
	VAR speeddata vd393 :=[6.76,500,5000,2.38];
	VAR speeddata vd394 :=[6.82,500,5000,2.35];
	VAR speeddata vd395 :=[6.87,500,5000,2.31];
	VAR speeddata vd396 :=[6.93,500,5000,2.28];
	VAR speeddata vd397 :=[6.99,500,5000,2.24];
	VAR speeddata vd398 :=[7.04,500,5000,2.21];
	VAR speeddata vd399 :=[7.04,500,5000,2.21];
	VAR speeddata vd400 :=[6.99,500,5000,2.24];
	VAR speeddata vd401 :=[6.93,500,5000,2.28];
	VAR speeddata vd402 :=[6.87,500,5000,2.31];
	VAR speeddata vd403 :=[6.82,500,5000,2.35];
	VAR speeddata vd404 :=[6.76,500,5000,2.38];
	VAR speeddata vd405 :=[6.69,500,5000,2.42];
	VAR speeddata vd406 :=[6.63,500,5000,2.45];
	VAR speeddata vd407 :=[6.56,500,5000,2.49];
	VAR speeddata vd408 :=[6.50,500,5000,2.53];
	VAR speeddata vd409 :=[6.43,500,5000,2.57];
	VAR speeddata vd410 :=[6.36,500,5000,2.61];
	VAR speeddata vd411 :=[6.29,500,5000,2.65];
	VAR speeddata vd412 :=[6.22,500,5000,2.69];
	VAR speeddata vd413 :=[6.14,500,5000,2.73];
	VAR speeddata vd414 :=[6.07,500,5000,2.77];
	VAR speeddata vd415 :=[5.99,500,5000,2.81];
	VAR speeddata vd416 :=[5.91,500,5000,2.85];
	VAR speeddata vd417 :=[5.83,500,5000,2.89];
	VAR speeddata vd418 :=[5.75,500,5000,2.93];
	VAR speeddata vd419 :=[5.66,500,5000,2.98];
	VAR speeddata vd420 :=[5.58,500,5000,3.02];
	VAR speeddata vd421 :=[5.49,500,5000,3.06];
	VAR speeddata vd422 :=[5.40,500,5000,3.10];
	VAR speeddata vd423 :=[5.31,500,5000,3.15];
	VAR speeddata vd424 :=[5.21,500,5000,3.19];
	VAR speeddata vd425 :=[5.12,500,5000,3.23];
	VAR speeddata vd426 :=[5.02,500,5000,3.28];
	VAR speeddata vd427 :=[4.92,500,5000,3.32];
	VAR speeddata vd428 :=[4.82,500,5000,3.36];
	VAR speeddata vd429 :=[4.71,500,5000,3.41];
	VAR speeddata vd430 :=[4.61,500,5000,3.45];
	VAR speeddata vd431 :=[4.50,500,5000,3.49];
	VAR speeddata vd432 :=[4.39,500,5000,3.54];
	VAR speeddata vd433 :=[4.28,500,5000,3.58];
	VAR speeddata vd434 :=[4.16,500,5000,3.62];
	VAR speeddata vd435 :=[4.05,500,5000,3.66];
	VAR speeddata vd436 :=[3.93,500,5000,3.70];
	VAR speeddata vd437 :=[3.81,500,5000,3.74];
	VAR speeddata vd438 :=[3.69,500,5000,3.78];
	VAR speeddata vd439 :=[3.57,500,5000,3.82];
	VAR speeddata vd440 :=[3.44,500,5000,3.86];
	VAR speeddata vd441 :=[3.31,500,5000,3.90];
	VAR speeddata vd442 :=[3.19,500,5000,3.94];
	VAR speeddata vd443 :=[3.05,500,5000,3.97];
	VAR speeddata vd444 :=[2.92,500,5000,4.01];
	VAR speeddata vd445 :=[2.79,500,5000,4.04];
	VAR speeddata vd446 :=[2.65,500,5000,4.07];
	VAR speeddata vd447 :=[2.51,500,5000,4.10];
	VAR speeddata vd448 :=[2.37,500,5000,4.13];
	VAR speeddata vd449 :=[2.23,500,5000,4.16];
	VAR speeddata vd450 :=[2.09,500,5000,4.19];
	VAR speeddata vd451 :=[1.95,500,5000,4.21];
	VAR speeddata vd452 :=[1.80,500,5000,4.24];
	VAR speeddata vd453 :=[1.66,500,5000,4.26];
	VAR speeddata vd454 :=[1.51,500,5000,4.28];
	VAR speeddata vd455 :=[1.36,500,5000,4.30];
	VAR speeddata vd456 :=[1.22,500,5000,4.32];
	VAR speeddata vd457 :=[1.07,500,5000,4.33];
	VAR speeddata vd458 :=[0.92,500,5000,4.34];
	VAR speeddata vd459 :=[0.77,500,5000,4.35];
	VAR speeddata vd460 :=[0.62,500,5000,4.36];
	VAR speeddata vd461 :=[0.47,500,5000,4.37];
	VAR speeddata vd462 :=[0.32,500,5000,4.38];
	VAR speeddata vd463 :=[0.18,500,5000,4.38];
	VAR speeddata vd464 :=[0.10,500,5000,4.38];
	VAR speeddata vd465 :=[0.18,500,5000,4.38];
	VAR speeddata vd466 :=[0.32,500,5000,4.38];
	VAR speeddata vd467 :=[0.47,500,5000,4.37];
	VAR speeddata vd468 :=[0.62,500,5000,4.36];
	VAR speeddata vd469 :=[0.77,500,5000,4.35];
	VAR speeddata vd470 :=[0.92,500,5000,4.34];
	VAR speeddata vd471 :=[1.07,500,5000,4.33];
	VAR speeddata vd472 :=[1.22,500,5000,4.32];
	VAR speeddata vd473 :=[1.36,500,5000,4.30];
	VAR speeddata vd474 :=[1.51,500,5000,4.28];
	VAR speeddata vd475 :=[1.66,500,5000,4.26];
	VAR speeddata vd476 :=[1.80,500,5000,4.24];
	VAR speeddata vd477 :=[1.95,500,5000,4.21];
	VAR speeddata vd478 :=[2.09,500,5000,4.19];
	VAR speeddata vd479 :=[2.23,500,5000,4.16];
	VAR speeddata vd480 :=[2.37,500,5000,4.13];
	VAR speeddata vd481 :=[2.51,500,5000,4.10];
	VAR speeddata vd482 :=[2.65,500,5000,4.07];
	VAR speeddata vd483 :=[2.79,500,5000,4.04];
	VAR speeddata vd484 :=[2.92,500,5000,4.01];
	VAR speeddata vd485 :=[3.05,500,5000,3.97];
	VAR speeddata vd486 :=[3.19,500,5000,3.94];
	VAR speeddata vd487 :=[3.31,500,5000,3.90];
	VAR speeddata vd488 :=[3.44,500,5000,3.86];
	VAR speeddata vd489 :=[3.57,500,5000,3.82];
	VAR speeddata vd490 :=[3.69,500,5000,3.78];
	VAR speeddata vd491 :=[3.81,500,5000,3.74];
	VAR speeddata vd492 :=[3.93,500,5000,3.70];
	VAR speeddata vd493 :=[4.05,500,5000,3.66];
	VAR speeddata vd494 :=[4.16,500,5000,3.62];
	VAR speeddata vd495 :=[4.28,500,5000,3.58];
	VAR speeddata vd496 :=[4.39,500,5000,3.54];
	VAR speeddata vd497 :=[4.50,500,5000,3.49];
	VAR speeddata vd498 :=[4.61,500,5000,3.45];
	VAR speeddata vd499 :=[4.71,500,5000,3.41];
	VAR speeddata vd500 :=[4.82,500,5000,3.36];
	VAR speeddata vd501 :=[4.92,500,5000,3.32];
	VAR speeddata vd502 :=[5.02,500,5000,3.28];
	VAR speeddata vd503 :=[5.12,500,5000,3.23];
	VAR speeddata vd504 :=[5.21,500,5000,3.19];
	VAR speeddata vd505 :=[5.31,500,5000,3.15];
	VAR speeddata vd506 :=[5.40,500,5000,3.10];
	VAR speeddata vd507 :=[5.49,500,5000,3.06];
	VAR speeddata vd508 :=[5.58,500,5000,3.02];
	VAR speeddata vd509 :=[5.66,500,5000,2.98];
	VAR speeddata vd510 :=[5.75,500,5000,2.93];
	VAR speeddata vd511 :=[5.83,500,5000,2.89];
	VAR speeddata vd512 :=[5.91,500,5000,2.85];
	VAR speeddata vd513 :=[5.99,500,5000,2.81];
	VAR speeddata vd514 :=[6.07,500,5000,2.77];
	VAR speeddata vd515 :=[6.14,500,5000,2.73];
	VAR speeddata vd516 :=[6.22,500,5000,2.69];
	VAR speeddata vd517 :=[6.29,500,5000,2.65];
	VAR speeddata vd518 :=[6.36,500,5000,2.61];
	VAR speeddata vd519 :=[6.43,500,5000,2.57];
	VAR speeddata vd520 :=[6.50,500,5000,2.53];
	VAR speeddata vd521 :=[6.56,500,5000,2.49];
	VAR speeddata vd522 :=[6.63,500,5000,2.45];
	VAR speeddata vd523 :=[6.69,500,5000,2.42];
	VAR speeddata vd524 :=[6.76,500,5000,2.38];
	VAR speeddata vd525 :=[6.82,500,5000,2.35];
	VAR speeddata vd526 :=[6.87,500,5000,2.31];
	VAR speeddata vd527 :=[6.93,500,5000,2.28];
	VAR speeddata vd528 :=[6.99,500,5000,2.24];
	VAR speeddata vd529 :=[7.04,500,5000,2.21];
	VAR speeddata vd530 :=[7.14,500,5000,2.18];
	VAR speeddata vd531 :=[7.09,500,5000,2.21];
	VAR speeddata vd532 :=[7.03,500,5000,2.24];
	VAR speeddata vd533 :=[6.98,500,5000,2.28];
	VAR speeddata vd534 :=[6.92,500,5000,2.31];
	VAR speeddata vd535 :=[6.86,500,5000,2.35];
	VAR speeddata vd536 :=[6.80,500,5000,2.39];
	VAR speeddata vd537 :=[6.74,500,5000,2.42];
	VAR speeddata vd538 :=[6.68,500,5000,2.46];
	VAR speeddata vd539 :=[6.61,500,5000,2.50];
	VAR speeddata vd540 :=[6.55,500,5000,2.54];
	VAR speeddata vd541 :=[6.48,500,5000,2.58];
	VAR speeddata vd542 :=[6.41,500,5000,2.62];
	VAR speeddata vd543 :=[6.34,500,5000,2.66];
	VAR speeddata vd544 :=[6.27,500,5000,2.70];
	VAR speeddata vd545 :=[6.20,500,5000,2.74];
	VAR speeddata vd546 :=[6.12,500,5000,2.78];
	VAR speeddata vd547 :=[6.04,500,5000,2.82];
	VAR speeddata vd548 :=[5.96,500,5000,2.86];
	VAR speeddata vd549 :=[5.88,500,5000,2.90];
	VAR speeddata vd550 :=[5.80,500,5000,2.95];
	VAR speeddata vd551 :=[5.72,500,5000,2.99];
	VAR speeddata vd552 :=[5.63,500,5000,3.03];
	VAR speeddata vd553 :=[5.54,500,5000,3.08];
	VAR speeddata vd554 :=[5.45,500,5000,3.12];
	VAR speeddata vd555 :=[5.36,500,5000,3.16];
	VAR speeddata vd556 :=[5.27,500,5000,3.21];
	VAR speeddata vd557 :=[5.17,500,5000,3.25];
	VAR speeddata vd558 :=[5.08,500,5000,3.30];
	VAR speeddata vd559 :=[4.98,500,5000,3.34];
	VAR speeddata vd560 :=[4.88,500,5000,3.39];
	VAR speeddata vd561 :=[4.77,500,5000,3.43];
	VAR speeddata vd562 :=[4.67,500,5000,3.47];
	VAR speeddata vd563 :=[4.56,500,5000,3.52];
	VAR speeddata vd564 :=[4.45,500,5000,3.56];
	VAR speeddata vd565 :=[4.34,500,5000,3.61];
	VAR speeddata vd566 :=[4.22,500,5000,3.65];
	VAR speeddata vd567 :=[4.11,500,5000,3.69];
	VAR speeddata vd568 :=[3.99,500,5000,3.73];
	VAR speeddata vd569 :=[3.87,500,5000,3.78];
	VAR speeddata vd570 :=[3.75,500,5000,3.82];
	VAR speeddata vd571 :=[3.63,500,5000,3.86];
	VAR speeddata vd572 :=[3.50,500,5000,3.90];
	VAR speeddata vd573 :=[3.37,500,5000,3.94];
	VAR speeddata vd574 :=[3.24,500,5000,3.97];
	VAR speeddata vd575 :=[3.11,500,5000,4.01];
	VAR speeddata vd576 :=[2.98,500,5000,4.05];
	VAR speeddata vd577 :=[2.85,500,5000,4.08];
	VAR speeddata vd578 :=[2.71,500,5000,4.12];
	VAR speeddata vd579 :=[2.57,500,5000,4.15];
	VAR speeddata vd580 :=[2.43,500,5000,4.18];
	VAR speeddata vd581 :=[2.29,500,5000,4.21];
	VAR speeddata vd582 :=[2.15,500,5000,4.24];
	VAR speeddata vd583 :=[2.00,500,5000,4.26];
	VAR speeddata vd584 :=[1.86,500,5000,4.29];
	VAR speeddata vd585 :=[1.71,500,5000,4.31];
	VAR speeddata vd586 :=[1.57,500,5000,4.33];
	VAR speeddata vd587 :=[1.42,500,5000,4.35];
	VAR speeddata vd588 :=[1.27,500,5000,4.37];
	VAR speeddata vd589 :=[1.12,500,5000,4.39];
	VAR speeddata vd590 :=[0.97,500,5000,4.40];
	VAR speeddata vd591 :=[0.82,500,5000,4.41];
	VAR speeddata vd592 :=[0.66,500,5000,4.42];
	VAR speeddata vd593 :=[0.51,500,5000,4.43];
	VAR speeddata vd594 :=[0.36,500,5000,4.44];
	VAR speeddata vd595 :=[0.22,500,5000,4.44];
	VAR speeddata vd596 :=[0.11,500,5000,4.44];
	VAR speeddata vd597 :=[0.15,500,5000,4.44];
	VAR speeddata vd598 :=[0.28,500,5000,4.44];
	VAR speeddata vd599 :=[0.43,500,5000,4.43];
	VAR speeddata vd600 :=[0.58,500,5000,4.43];
	VAR speeddata vd601 :=[0.73,500,5000,4.42];
	VAR speeddata vd602 :=[0.88,500,5000,4.41];
	VAR speeddata vd603 :=[1.03,500,5000,4.39];
	VAR speeddata vd604 :=[1.18,500,5000,4.38];
	VAR speeddata vd605 :=[1.33,500,5000,4.36];
	VAR speeddata vd606 :=[1.48,500,5000,4.34];
	VAR speeddata vd607 :=[1.63,500,5000,4.32];
	VAR speeddata vd608 :=[1.78,500,5000,4.30];
	VAR speeddata vd609 :=[1.92,500,5000,4.28];
	VAR speeddata vd610 :=[2.07,500,5000,4.25];
	VAR speeddata vd611 :=[2.21,500,5000,4.22];
	VAR speeddata vd612 :=[2.35,500,5000,4.20];
	VAR speeddata vd613 :=[2.49,500,5000,4.17];
	VAR speeddata vd614 :=[2.63,500,5000,4.13];
	VAR speeddata vd615 :=[2.77,500,5000,4.10];
	VAR speeddata vd616 :=[2.91,500,5000,4.07];
	VAR speeddata vd617 :=[3.04,500,5000,4.03];
	VAR speeddata vd618 :=[3.17,500,5000,3.99];
	VAR speeddata vd619 :=[3.30,500,5000,3.96];
	VAR speeddata vd620 :=[3.43,500,5000,3.92];
	VAR speeddata vd621 :=[3.56,500,5000,3.88];
	VAR speeddata vd622 :=[3.68,500,5000,3.84];
	VAR speeddata vd623 :=[3.80,500,5000,3.80];
	VAR speeddata vd624 :=[3.92,500,5000,3.76];
	VAR speeddata vd625 :=[4.04,500,5000,3.72];
	VAR speeddata vd626 :=[4.16,500,5000,3.67];
	VAR speeddata vd627 :=[4.28,500,5000,3.63];
	VAR speeddata vd628 :=[4.39,500,5000,3.59];
	VAR speeddata vd629 :=[4.50,500,5000,3.54];
	VAR speeddata vd630 :=[4.61,500,5000,3.50];
	VAR speeddata vd631 :=[4.71,500,5000,3.45];
	VAR speeddata vd632 :=[4.82,500,5000,3.41];
	VAR speeddata vd633 :=[4.92,500,5000,3.37];
	VAR speeddata vd634 :=[5.02,500,5000,3.32];
	VAR speeddata vd635 :=[5.12,500,5000,3.28];
	VAR speeddata vd636 :=[5.22,500,5000,3.23];
	VAR speeddata vd637 :=[5.31,500,5000,3.19];
	VAR speeddata vd638 :=[5.40,500,5000,3.14];
	VAR speeddata vd639 :=[5.49,500,5000,3.10];
	VAR speeddata vd640 :=[5.58,500,5000,3.06];
	VAR speeddata vd641 :=[5.67,500,5000,3.01];
	VAR speeddata vd642 :=[5.76,500,5000,2.97];
	VAR speeddata vd643 :=[5.84,500,5000,2.93];
	VAR speeddata vd644 :=[5.92,500,5000,2.88];
	VAR speeddata vd645 :=[6.00,500,5000,2.84];
	VAR speeddata vd646 :=[6.08,500,5000,2.80];
	VAR speeddata vd647 :=[6.15,500,5000,2.76];
	VAR speeddata vd648 :=[6.23,500,5000,2.72];
	VAR speeddata vd649 :=[6.30,500,5000,2.68];
	VAR speeddata vd650 :=[6.37,500,5000,2.64];
	VAR speeddata vd651 :=[6.44,500,5000,2.60];
	VAR speeddata vd652 :=[6.51,500,5000,2.56];
	VAR speeddata vd653 :=[6.58,500,5000,2.52];
	VAR speeddata vd654 :=[6.64,500,5000,2.48];
	VAR speeddata vd655 :=[6.71,500,5000,2.44];
	VAR speeddata vd656 :=[6.77,500,5000,2.41];
	VAR speeddata vd657 :=[6.83,500,5000,2.37];
	VAR speeddata vd658 :=[6.89,500,5000,2.33];
	VAR speeddata vd659 :=[6.95,500,5000,2.30];
	VAR speeddata vd660 :=[7.04,500,5000,2.27];
	VAR speeddata vd661 :=[6.99,500,5000,2.30];
	VAR speeddata vd662 :=[6.93,500,5000,2.34];
	VAR speeddata vd663 :=[6.87,500,5000,2.38];
	VAR speeddata vd664 :=[6.81,500,5000,2.41];
	VAR speeddata vd665 :=[6.75,500,5000,2.45];
	VAR speeddata vd666 :=[6.68,500,5000,2.49];
	VAR speeddata vd667 :=[6.62,500,5000,2.53];
	VAR speeddata vd668 :=[6.55,500,5000,2.57];
	VAR speeddata vd669 :=[6.48,500,5000,2.61];
	VAR speeddata vd670 :=[6.41,500,5000,2.65];
	VAR speeddata vd671 :=[6.34,500,5000,2.69];
	VAR speeddata vd672 :=[6.27,500,5000,2.73];
	VAR speeddata vd673 :=[6.19,500,5000,2.77];
	VAR speeddata vd674 :=[6.12,500,5000,2.82];
	VAR speeddata vd675 :=[6.04,500,5000,2.86];
	VAR speeddata vd676 :=[5.96,500,5000,2.90];
	VAR speeddata vd677 :=[5.88,500,5000,2.95];
	VAR speeddata vd678 :=[5.79,500,5000,2.99];
	VAR speeddata vd679 :=[5.71,500,5000,3.03];
	VAR speeddata vd680 :=[5.62,500,5000,3.08];
	VAR speeddata vd681 :=[5.53,500,5000,3.12];
	VAR speeddata vd682 :=[5.44,500,5000,3.17];
	VAR speeddata vd683 :=[5.35,500,5000,3.21];
	VAR speeddata vd684 :=[5.25,500,5000,3.26];
	VAR speeddata vd685 :=[5.16,500,5000,3.31];
	VAR speeddata vd686 :=[5.06,500,5000,3.35];
	VAR speeddata vd687 :=[4.95,500,5000,3.40];
	VAR speeddata vd688 :=[4.85,500,5000,3.44];
	VAR speeddata vd689 :=[4.75,500,5000,3.49];
	VAR speeddata vd690 :=[4.64,500,5000,3.53];
	VAR speeddata vd691 :=[4.53,500,5000,3.58];
	VAR speeddata vd692 :=[4.42,500,5000,3.62];
	VAR speeddata vd693 :=[4.30,500,5000,3.67];
	VAR speeddata vd694 :=[4.19,500,5000,3.71];
	VAR speeddata vd695 :=[4.07,500,5000,3.76];
	VAR speeddata vd696 :=[3.95,500,5000,3.80];
	VAR speeddata vd697 :=[3.83,500,5000,3.84];
	VAR speeddata vd698 :=[3.70,500,5000,3.88];
	VAR speeddata vd699 :=[3.58,500,5000,3.93];
	VAR speeddata vd700 :=[3.45,500,5000,3.97];
	VAR speeddata vd701 :=[3.32,500,5000,4.01];
	VAR speeddata vd702 :=[3.19,500,5000,4.04];
	VAR speeddata vd703 :=[3.05,500,5000,4.08];
	VAR speeddata vd704 :=[2.92,500,5000,4.12];
	VAR speeddata vd705 :=[2.78,500,5000,4.15];
	VAR speeddata vd706 :=[2.64,500,5000,4.19];
	VAR speeddata vd707 :=[2.50,500,5000,4.22];
	VAR speeddata vd708 :=[2.36,500,5000,4.25];
	VAR speeddata vd709 :=[2.21,500,5000,4.28];
	VAR speeddata vd710 :=[2.07,500,5000,4.31];
	VAR speeddata vd711 :=[1.92,500,5000,4.34];
	VAR speeddata vd712 :=[1.77,500,5000,4.36];
	VAR speeddata vd713 :=[1.62,500,5000,4.38];
	VAR speeddata vd714 :=[1.47,500,5000,4.40];
	VAR speeddata vd715 :=[1.32,500,5000,4.42];
	VAR speeddata vd716 :=[1.17,500,5000,4.44];
	VAR speeddata vd717 :=[1.02,500,5000,4.46];
	VAR speeddata vd718 :=[0.86,500,5000,4.47];
	VAR speeddata vd719 :=[0.71,500,5000,4.48];
	VAR speeddata vd720 :=[0.55,500,5000,4.49];
	VAR speeddata vd721 :=[0.40,500,5000,4.49];
	VAR speeddata vd722 :=[0.25,500,5000,4.50];
	VAR speeddata vd723 :=[0.13,500,5000,4.50];
	VAR speeddata vd724 :=[0.13,500,5000,4.50];
	VAR speeddata vd725 :=[0.25,500,5000,4.50];
	VAR speeddata vd726 :=[0.40,500,5000,4.49];
	VAR speeddata vd727 :=[0.55,500,5000,4.49];
	VAR speeddata vd728 :=[0.71,500,5000,4.48];
	VAR speeddata vd729 :=[0.86,500,5000,4.47];
	VAR speeddata vd730 :=[1.02,500,5000,4.46];
	VAR speeddata vd731 :=[1.17,500,5000,4.44];
	VAR speeddata vd732 :=[1.32,500,5000,4.42];
	VAR speeddata vd733 :=[1.47,500,5000,4.40];
	VAR speeddata vd734 :=[1.62,500,5000,4.38];
	VAR speeddata vd735 :=[1.77,500,5000,4.36];
	VAR speeddata vd736 :=[1.92,500,5000,4.34];
	VAR speeddata vd737 :=[2.07,500,5000,4.31];
	VAR speeddata vd738 :=[2.21,500,5000,4.28];
	VAR speeddata vd739 :=[2.36,500,5000,4.25];
	VAR speeddata vd740 :=[2.50,500,5000,4.22];
	VAR speeddata vd741 :=[2.64,500,5000,4.19];
	VAR speeddata vd742 :=[2.78,500,5000,4.15];
	VAR speeddata vd743 :=[2.92,500,5000,4.12];
	VAR speeddata vd744 :=[3.05,500,5000,4.08];
	VAR speeddata vd745 :=[3.19,500,5000,4.04];
	VAR speeddata vd746 :=[3.32,500,5000,4.01];
	VAR speeddata vd747 :=[3.45,500,5000,3.97];
	VAR speeddata vd748 :=[3.58,500,5000,3.93];
	VAR speeddata vd749 :=[3.70,500,5000,3.88];
	VAR speeddata vd750 :=[3.83,500,5000,3.84];
	VAR speeddata vd751 :=[3.95,500,5000,3.80];
	VAR speeddata vd752 :=[4.07,500,5000,3.76];
	VAR speeddata vd753 :=[4.19,500,5000,3.71];
	VAR speeddata vd754 :=[4.30,500,5000,3.67];
	VAR speeddata vd755 :=[4.42,500,5000,3.62];
	VAR speeddata vd756 :=[4.53,500,5000,3.58];
	VAR speeddata vd757 :=[4.64,500,5000,3.53];
	VAR speeddata vd758 :=[4.75,500,5000,3.49];
	VAR speeddata vd759 :=[4.85,500,5000,3.44];
	VAR speeddata vd760 :=[4.95,500,5000,3.40];
	VAR speeddata vd761 :=[5.06,500,5000,3.35];
	VAR speeddata vd762 :=[5.16,500,5000,3.31];
	VAR speeddata vd763 :=[5.25,500,5000,3.26];
	VAR speeddata vd764 :=[5.35,500,5000,3.21];
	VAR speeddata vd765 :=[5.44,500,5000,3.17];
	VAR speeddata vd766 :=[5.53,500,5000,3.12];
	VAR speeddata vd767 :=[5.62,500,5000,3.08];
	VAR speeddata vd768 :=[5.71,500,5000,3.03];
	VAR speeddata vd769 :=[5.79,500,5000,2.99];
	VAR speeddata vd770 :=[5.88,500,5000,2.95];
	VAR speeddata vd771 :=[5.96,500,5000,2.90];
	VAR speeddata vd772 :=[6.04,500,5000,2.86];
	VAR speeddata vd773 :=[6.12,500,5000,2.82];
	VAR speeddata vd774 :=[6.19,500,5000,2.77];
	VAR speeddata vd775 :=[6.27,500,5000,2.73];
	VAR speeddata vd776 :=[6.34,500,5000,2.69];
	VAR speeddata vd777 :=[6.41,500,5000,2.65];
	VAR speeddata vd778 :=[6.48,500,5000,2.61];
	VAR speeddata vd779 :=[6.55,500,5000,2.57];
	VAR speeddata vd780 :=[6.62,500,5000,2.53];
	VAR speeddata vd781 :=[6.68,500,5000,2.49];
	VAR speeddata vd782 :=[6.75,500,5000,2.45];
	VAR speeddata vd783 :=[6.81,500,5000,2.41];
	VAR speeddata vd784 :=[6.87,500,5000,2.38];
	VAR speeddata vd785 :=[6.93,500,5000,2.34];
	VAR speeddata vd786 :=[6.99,500,5000,2.30];
	VAR speeddata vd787 :=[7.04,500,5000,2.27];
	VAR speeddata vd788 :=[7.04,500,5000,2.27];
	VAR speeddata vd789 :=[6.99,500,5000,2.30];
	VAR speeddata vd790 :=[6.93,500,5000,2.34];
	VAR speeddata vd791 :=[6.87,500,5000,2.38];
	VAR speeddata vd792 :=[6.81,500,5000,2.41];
	VAR speeddata vd793 :=[6.75,500,5000,2.45];
	VAR speeddata vd794 :=[6.68,500,5000,2.49];
	VAR speeddata vd795 :=[6.62,500,5000,2.53];
	VAR speeddata vd796 :=[6.55,500,5000,2.57];
	VAR speeddata vd797 :=[6.48,500,5000,2.61];
	VAR speeddata vd798 :=[6.41,500,5000,2.65];
	VAR speeddata vd799 :=[6.34,500,5000,2.69];
	VAR speeddata vd800 :=[6.27,500,5000,2.73];
	VAR speeddata vd801 :=[6.19,500,5000,2.77];
	VAR speeddata vd802 :=[6.12,500,5000,2.82];
	VAR speeddata vd803 :=[6.04,500,5000,2.86];
	VAR speeddata vd804 :=[5.96,500,5000,2.90];
	VAR speeddata vd805 :=[5.88,500,5000,2.95];
	VAR speeddata vd806 :=[5.79,500,5000,2.99];
	VAR speeddata vd807 :=[5.71,500,5000,3.03];
	VAR speeddata vd808 :=[5.62,500,5000,3.08];
	VAR speeddata vd809 :=[5.53,500,5000,3.12];
	VAR speeddata vd810 :=[5.44,500,5000,3.17];
	VAR speeddata vd811 :=[5.35,500,5000,3.21];
	VAR speeddata vd812 :=[5.25,500,5000,3.26];
	VAR speeddata vd813 :=[5.16,500,5000,3.31];
	VAR speeddata vd814 :=[5.06,500,5000,3.35];
	VAR speeddata vd815 :=[4.95,500,5000,3.40];
	VAR speeddata vd816 :=[4.85,500,5000,3.44];
	VAR speeddata vd817 :=[4.75,500,5000,3.49];
	VAR speeddata vd818 :=[4.64,500,5000,3.53];
	VAR speeddata vd819 :=[4.53,500,5000,3.58];
	VAR speeddata vd820 :=[4.42,500,5000,3.62];
	VAR speeddata vd821 :=[4.30,500,5000,3.67];
	VAR speeddata vd822 :=[4.19,500,5000,3.71];
	VAR speeddata vd823 :=[4.07,500,5000,3.76];
	VAR speeddata vd824 :=[3.95,500,5000,3.80];
	VAR speeddata vd825 :=[3.83,500,5000,3.84];
	VAR speeddata vd826 :=[3.70,500,5000,3.88];
	VAR speeddata vd827 :=[3.58,500,5000,3.93];
	VAR speeddata vd828 :=[3.45,500,5000,3.97];
	VAR speeddata vd829 :=[3.32,500,5000,4.01];
	VAR speeddata vd830 :=[3.19,500,5000,4.04];
	VAR speeddata vd831 :=[3.05,500,5000,4.08];
	VAR speeddata vd832 :=[2.92,500,5000,4.12];
	VAR speeddata vd833 :=[2.78,500,5000,4.15];
	VAR speeddata vd834 :=[2.64,500,5000,4.19];
	VAR speeddata vd835 :=[2.50,500,5000,4.22];
	VAR speeddata vd836 :=[2.36,500,5000,4.25];
	VAR speeddata vd837 :=[2.21,500,5000,4.28];
	VAR speeddata vd838 :=[2.07,500,5000,4.31];
	VAR speeddata vd839 :=[1.92,500,5000,4.34];
	VAR speeddata vd840 :=[1.77,500,5000,4.36];
	VAR speeddata vd841 :=[1.62,500,5000,4.38];
	VAR speeddata vd842 :=[1.47,500,5000,4.40];
	VAR speeddata vd843 :=[1.32,500,5000,4.42];
	VAR speeddata vd844 :=[1.17,500,5000,4.44];
	VAR speeddata vd845 :=[1.02,500,5000,4.46];
	VAR speeddata vd846 :=[0.86,500,5000,4.47];
	VAR speeddata vd847 :=[0.71,500,5000,4.48];
	VAR speeddata vd848 :=[0.55,500,5000,4.49];
	VAR speeddata vd849 :=[0.40,500,5000,4.49];
	VAR speeddata vd850 :=[0.25,500,5000,4.50];
	VAR speeddata vd851 :=[0.13,500,5000,4.50];
	VAR speeddata vd852 :=[0.13,500,5000,4.50];
	VAR speeddata vd853 :=[0.25,500,5000,4.50];
	VAR speeddata vd854 :=[0.40,500,5000,4.49];
	VAR speeddata vd855 :=[0.55,500,5000,4.49];
	VAR speeddata vd856 :=[0.71,500,5000,4.48];
	VAR speeddata vd857 :=[0.86,500,5000,4.47];
	VAR speeddata vd858 :=[1.02,500,5000,4.46];
	VAR speeddata vd859 :=[1.17,500,5000,4.44];
	VAR speeddata vd860 :=[1.32,500,5000,4.42];
	VAR speeddata vd861 :=[1.47,500,5000,4.40];
	VAR speeddata vd862 :=[1.62,500,5000,4.38];
	VAR speeddata vd863 :=[1.77,500,5000,4.36];
	VAR speeddata vd864 :=[1.92,500,5000,4.34];
	VAR speeddata vd865 :=[2.07,500,5000,4.31];
	VAR speeddata vd866 :=[2.21,500,5000,4.28];
	VAR speeddata vd867 :=[2.36,500,5000,4.25];
	VAR speeddata vd868 :=[2.50,500,5000,4.22];
	VAR speeddata vd869 :=[2.64,500,5000,4.19];
	VAR speeddata vd870 :=[2.78,500,5000,4.15];
	VAR speeddata vd871 :=[2.92,500,5000,4.12];
	VAR speeddata vd872 :=[3.05,500,5000,4.08];
	VAR speeddata vd873 :=[3.19,500,5000,4.04];
	VAR speeddata vd874 :=[3.32,500,5000,4.01];
	VAR speeddata vd875 :=[3.45,500,5000,3.97];
	VAR speeddata vd876 :=[3.58,500,5000,3.93];
	VAR speeddata vd877 :=[3.70,500,5000,3.88];
	VAR speeddata vd878 :=[3.83,500,5000,3.84];
	VAR speeddata vd879 :=[3.95,500,5000,3.80];
	VAR speeddata vd880 :=[4.07,500,5000,3.76];
	VAR speeddata vd881 :=[4.19,500,5000,3.71];
	VAR speeddata vd882 :=[4.30,500,5000,3.67];
	VAR speeddata vd883 :=[4.42,500,5000,3.62];
	VAR speeddata vd884 :=[4.53,500,5000,3.58];
	VAR speeddata vd885 :=[4.64,500,5000,3.53];
	VAR speeddata vd886 :=[4.75,500,5000,3.49];
	VAR speeddata vd887 :=[4.85,500,5000,3.44];
	VAR speeddata vd888 :=[4.95,500,5000,3.40];
	VAR speeddata vd889 :=[5.06,500,5000,3.35];
	VAR speeddata vd890 :=[5.16,500,5000,3.31];
	VAR speeddata vd891 :=[5.25,500,5000,3.26];
	VAR speeddata vd892 :=[5.35,500,5000,3.21];
	VAR speeddata vd893 :=[5.44,500,5000,3.17];
	VAR speeddata vd894 :=[5.53,500,5000,3.12];
	VAR speeddata vd895 :=[5.62,500,5000,3.08];
	VAR speeddata vd896 :=[5.71,500,5000,3.03];
	VAR speeddata vd897 :=[5.79,500,5000,2.99];
	VAR speeddata vd898 :=[5.88,500,5000,2.95];
	VAR speeddata vd899 :=[5.96,500,5000,2.90];
	VAR speeddata vd900 :=[6.04,500,5000,2.86];
	VAR speeddata vd901 :=[6.12,500,5000,2.82];
	VAR speeddata vd902 :=[6.19,500,5000,2.77];
	VAR speeddata vd903 :=[6.27,500,5000,2.73];
	VAR speeddata vd904 :=[6.34,500,5000,2.69];
	VAR speeddata vd905 :=[6.41,500,5000,2.65];
	VAR speeddata vd906 :=[6.48,500,5000,2.61];
	VAR speeddata vd907 :=[6.55,500,5000,2.57];
	VAR speeddata vd908 :=[6.62,500,5000,2.53];
	VAR speeddata vd909 :=[6.68,500,5000,2.49];
	VAR speeddata vd910 :=[6.75,500,5000,2.45];
	VAR speeddata vd911 :=[6.81,500,5000,2.41];
	VAR speeddata vd912 :=[6.87,500,5000,2.38];
	VAR speeddata vd913 :=[6.93,500,5000,2.34];
	VAR speeddata vd914 :=[6.99,500,5000,2.30];
	VAR speeddata vd915 :=[7.04,500,5000,2.27];
	VAR speeddata vd916 :=[7.04,500,5000,2.27];
	VAR speeddata vd917 :=[6.99,500,5000,2.30];
	VAR speeddata vd918 :=[6.93,500,5000,2.34];
	VAR speeddata vd919 :=[6.87,500,5000,2.38];
	VAR speeddata vd920 :=[6.81,500,5000,2.41];
	VAR speeddata vd921 :=[6.75,500,5000,2.45];
	VAR speeddata vd922 :=[6.68,500,5000,2.49];
	VAR speeddata vd923 :=[6.62,500,5000,2.53];
	VAR speeddata vd924 :=[6.55,500,5000,2.57];
	VAR speeddata vd925 :=[6.48,500,5000,2.61];
	VAR speeddata vd926 :=[6.41,500,5000,2.65];
	VAR speeddata vd927 :=[6.34,500,5000,2.69];
	VAR speeddata vd928 :=[6.27,500,5000,2.73];
	VAR speeddata vd929 :=[6.19,500,5000,2.77];
	VAR speeddata vd930 :=[6.12,500,5000,2.82];
	VAR speeddata vd931 :=[6.04,500,5000,2.86];
	VAR speeddata vd932 :=[5.96,500,5000,2.90];
	VAR speeddata vd933 :=[5.88,500,5000,2.95];
	VAR speeddata vd934 :=[5.79,500,5000,2.99];
	VAR speeddata vd935 :=[5.71,500,5000,3.03];
	VAR speeddata vd936 :=[5.62,500,5000,3.08];
	VAR speeddata vd937 :=[5.53,500,5000,3.12];
	VAR speeddata vd938 :=[5.44,500,5000,3.17];
	VAR speeddata vd939 :=[5.35,500,5000,3.21];
	VAR speeddata vd940 :=[5.25,500,5000,3.26];
	VAR speeddata vd941 :=[5.16,500,5000,3.31];
	VAR speeddata vd942 :=[5.06,500,5000,3.35];
	VAR speeddata vd943 :=[4.95,500,5000,3.40];
	VAR speeddata vd944 :=[4.85,500,5000,3.44];
	VAR speeddata vd945 :=[4.75,500,5000,3.49];
	VAR speeddata vd946 :=[4.64,500,5000,3.53];
	VAR speeddata vd947 :=[4.53,500,5000,3.58];
	VAR speeddata vd948 :=[4.42,500,5000,3.62];
	VAR speeddata vd949 :=[4.30,500,5000,3.67];
	VAR speeddata vd950 :=[4.19,500,5000,3.71];
	VAR speeddata vd951 :=[4.07,500,5000,3.76];
	VAR speeddata vd952 :=[3.95,500,5000,3.80];
	VAR speeddata vd953 :=[3.83,500,5000,3.84];
	VAR speeddata vd954 :=[3.70,500,5000,3.88];
	VAR speeddata vd955 :=[3.58,500,5000,3.93];
	VAR speeddata vd956 :=[3.45,500,5000,3.97];
	VAR speeddata vd957 :=[3.32,500,5000,4.01];
	VAR speeddata vd958 :=[3.19,500,5000,4.04];
	VAR speeddata vd959 :=[3.05,500,5000,4.08];
	VAR speeddata vd960 :=[2.92,500,5000,4.12];
	VAR speeddata vd961 :=[2.78,500,5000,4.15];
	VAR speeddata vd962 :=[2.64,500,5000,4.19];
	VAR speeddata vd963 :=[2.50,500,5000,4.22];
	VAR speeddata vd964 :=[2.36,500,5000,4.25];
	VAR speeddata vd965 :=[2.21,500,5000,4.28];
	VAR speeddata vd966 :=[2.07,500,5000,4.31];
	VAR speeddata vd967 :=[1.92,500,5000,4.34];
	VAR speeddata vd968 :=[1.77,500,5000,4.36];
	VAR speeddata vd969 :=[1.62,500,5000,4.38];
	VAR speeddata vd970 :=[1.47,500,5000,4.40];
	VAR speeddata vd971 :=[1.32,500,5000,4.42];
	VAR speeddata vd972 :=[1.17,500,5000,4.44];
	VAR speeddata vd973 :=[1.02,500,5000,4.46];
	VAR speeddata vd974 :=[0.86,500,5000,4.47];
	VAR speeddata vd975 :=[0.71,500,5000,4.48];
	VAR speeddata vd976 :=[0.55,500,5000,4.49];
	VAR speeddata vd977 :=[0.40,500,5000,4.49];
	VAR speeddata vd978 :=[0.25,500,5000,4.50];
	VAR speeddata vd979 :=[0.13,500,5000,4.50];
	VAR speeddata vd980 :=[0.13,500,5000,4.50];
	VAR speeddata vd981 :=[0.25,500,5000,4.50];
	VAR speeddata vd982 :=[0.40,500,5000,4.49];
	VAR speeddata vd983 :=[0.55,500,5000,4.49];
	VAR speeddata vd984 :=[0.71,500,5000,4.48];
	VAR speeddata vd985 :=[0.86,500,5000,4.47];
	VAR speeddata vd986 :=[1.02,500,5000,4.46];
	VAR speeddata vd987 :=[1.17,500,5000,4.44];
	VAR speeddata vd988 :=[1.32,500,5000,4.42];
	VAR speeddata vd989 :=[1.47,500,5000,4.40];
	VAR speeddata vd990 :=[1.62,500,5000,4.38];
	VAR speeddata vd991 :=[1.77,500,5000,4.36];
	VAR speeddata vd992 :=[1.92,500,5000,4.34];
	VAR speeddata vd993 :=[2.07,500,5000,4.31];
	VAR speeddata vd994 :=[2.21,500,5000,4.28];
	VAR speeddata vd995 :=[2.36,500,5000,4.25];
	VAR speeddata vd996 :=[2.50,500,5000,4.22];
	VAR speeddata vd997 :=[2.64,500,5000,4.19];
	VAR speeddata vd998 :=[2.78,500,5000,4.15];
	VAR speeddata vd999 :=[2.92,500,5000,4.12];


    PROC stand()
        !set atribui 1 a variavel
        !reset atribui 0 a variavel


        reset doFr1RobotReady; ! O robo nao esta pronto para soldagem

        set doFr1OpMode2;   !seleciona tipo de soldagem TIG (110)
        set doFr1OpMode1;
        reset doFr1OpMode0;

        reset doFr1GasTest; !Abre (1) e fecha (0) a valvula de gas

        reset doFr1ColdWireDisable;  !(1) para desabilitar a alimentacao de arame e (0) para habilitar


        reset doFr1FeedForward;   !Para a alimentação de arame (caso acionado)
        reset doFr1FeedRetract;
        SetAO aoFr1WireSpeedWfi,400;! Define velocidade da alimentacao do arame [0-22000 mm/min]


        reset doFr1WeldingSim; ! Simulacao de solda

        reset doFr1DC_AC; !  AC (1) ou DC(0)
        set doFr1DCn_DCp; ! DC+ (1) ou DC- (0)

        set DoFr1PulseDisable; ! (1) para desabilitar funcao Pulsar e (0) para habilitar

        reset DoFr1PulseRange2;  ! Seleciona frequencia de pulsacao (vide manual)
        reset DoFr1PulseRange1;
        reset DoFr1PulseRange0;

        SetAO aoFr1Power,125; !Define a corrente principal do arco eletrico (0 a 500A)

        set doFr1DutyCycleDisable; ! (1)para desabilitar o Duty cycle e (0) para habilitar
        SetAO aoFr1DutyCycle, 255; ![0-255) varia o duty cycle de 10% a 90%
        SetAO aoFr1BaseCurrent,100;! A corrente de soldadagem é reduzida para 0 a 100% da corrente principal. [0 a 100]



        set doFr1ErrorReset; ! Reseta a memoria de erros
        WaitTime 0.5;
        reset doFr1ErrorReset;

    ENDPROC

    PROC start0()
        !set atribui 1 a variavel
        !reset atribui 0 a varaiavel


        !reset doFr1WeldingSim; ! Simulacao de solda

        set doFr1RobotReady; ! O robo esta pronto para soldagem

        set doFr1ErrorReset; ! Reseta a memoria de erros
        WaitTime 0.2;
        reset doFr1ErrorReset;

        set doFr1ArcOn;

        WaitDI diFr1ArcStable, 1;

        set doFr1FeedForward;   !Alimentação de arame (caso acionado)
        WaitTime 0.5;

    ENDPROC

    PROC stop0()
        !set atribui 1 a variavel
        !reset atribui 0 a varaiavel

        reset doFr1RobotReady; ! O robo nao esta pronto para soldagem
        reset doFr1FeedForward;   !Alimentação de arame (caso acionado)
        reset doFr1ArcOn;


    ENDPROC

    TRAP colision

        stop;
        StopMove;

    ENDTRAP


    PROC send_data()

        message:= "Mode;" + "auto";!NumToStr(area, 3);
        SocketSend socket1 \Str:=message;
        !WaitTime 0.01;
        SocketReceive socket1 \Str:= message;

        message:= "Execution;" + program_name;!NumToStr(area, 3);
        SocketSend socket1 \Str:=message;
        !WaitTime 0.01;
        SocketReceive socket1 \Str:= message;

        message:= "T;" + ValToStr(CTool());!NumToStr(area, 3);
        SocketSend socket1 \Str:=message;
        !WaitTime 0.01;
        SocketReceive socket1 \Str:= message;

        message:= "CW;" + ValToStr(CWobj());!NumToStr(area, 3);
        SocketSend socket1 \Str:=message;
        !WaitTime 0.01;
        SocketReceive socket1 \Str:= message;

        actual_pos:= CRobT(\Tool:=TTW5500_1 \WObj:=wobj1);
        !converted_boolean:=StrToVal(ValToStr(soTCPSpeed), converted_float);
        message:= "Speed;" + ValToStr(1000*AOutput(soTCPSpeed));!NumToStr(area, 3);
        SocketSend socket1 \Str:=message;
        !WaitTime 0.01;
        SocketReceive socket1 \Str:= message;

        message:= "MSpeed;" + ValToStr(MaxRobSpeed());!NumToStr(area, 3);
        SocketSend socket1 \Str:=message;
        !WaitTime 0.01;
        SocketReceive socket1 \Str:= message;

        message:= "RSpeed;" + ValToStr(CSpeedOverride());!NumToStr(area, 3);
        SocketSend socket1 \Str:=message;
        !WaitTime 0.01;
        SocketReceive socket1 \Str:= message;

        message:= "Welding;" + ValToStr(DOutput(doFr1ArcOn));!NumToStr(area, 3);
        SocketSend socket1 \Str:=message;
        !WaitTime 0.01;
        SocketReceive socket1 \Str:= message;

        message:= "WVoltage;" + ValToStr(AInput(aiFr1WeldingVoltage) + 16);!NumToStr(area, 3);
        SocketSend socket1 \Str:=message;
        !WaitTime 0.01;
        SocketReceive socket1 \Str:= message;

        message:= "WCurrent;" + ValToStr(AOutput(aoFr1Power));!NumToStr(area, 3);
        SocketSend socket1 \Str:=message;
        !WaitTime 0.01;
        SocketReceive socket1 \Str:= message;

        message:= "WSpeed;" + ValToStr(AOutput(aoFr1WireSpeedWfi));!NumToStr(area, 3);
        SocketSend socket1 \Str:=message;
        !WaitTime 0.01;
        SocketReceive socket1 \Str:= message;

        strTemp:=ValToStr(actual_pos.extax);
        message:= "PR;" + strTemp;!NumToStr(area, 3);
        SocketSend socket1 \Str:=message;
        !WaitTime 0.01;
        SocketReceive socket1 \Str:= message;

        strTemp:=ValToStr(actual_pos.trans) + "," + ValToStr(actual_pos.rot);
        message:= "CR;" + strTemp;!NumToStr(area, 3);
        SocketSend socket1 \Str:=message;
        !WaitTime 0.01;
        SocketReceive socket1 \Str:= message;

        message:= "Timestamp;" + CDate() + "," + CTime();!NumToStr(area, 3);
        SocketSend socket1 \Str:=message;
        SocketReceive socket1 \Str:= message;

        IF message = "Shutdown" THEN

            end_socket;

        ENDIF

    ENDPROC

    TRAP socket_management

        ISleep timeint;
        IF i = 1 THEN
            !127.0.0.1
            SocketCreate socket1;
            SocketConnect socket1, "127.0.0.1", 1884;
            SocketSend socket1 \Str:="Status;ONLINE";
            i:=2;
        ENDIF
        send_data;
        IF received_string = "Shutdown" THEN

            end_socket;

        ENDIF

        IWatch timeint;

    ENDTRAP

    PROC end_socket()

        IDelete timeint;
        send_data;
        SocketSend socket1 \Str:="Status;OFFLINE";
        SocketReceive socket1 \Str:= message;
        SocketClose socket1;

    ENDPROC

	PROC main()
        IEnable;
        i:=0;
        IF i = 0 THEN

            CONNECT timeint WITH socket_management;
            ITimer 0.1, timeint;
            i:=1;

        ENDIF


		!ActUnit STN1;
		Movej p1, vd1, z10, TTW5500_1 \WObj:=wobj1;
		stand;
		start0;

